(* Logix 5000 project; controller CarbonScout_MK6 vendor 1 type 14 code 154 rev 32.11; software revision 32.00; part 8 of 17 *)
(* tags used below, declared in another part *)
   AI_AIT_01 : P_AIn;   // pH
   AI_AIT_02 : P_AIn;   // DO
   AI_Booster : P_AIn;   // Booster Tank Level
   AI_FIT_01 : P_AIn;   // Purge water flow
   AI_LIT_01 : P_AIn;   // Carbon Scout Laser Level Transmitter
   AI_LIT_02 : P_AIn;   // Carbon Scout Cone Level Transmitter
   AI_PIT_01 : P_AIn;   // Water supply pressure
   AI_TIT_01 : P_AIn;   // Temperature
   AI_WIT_01 : P_AIn;   // Weight measure
   Client_to_Gekko : DINT[10];
   CS_Alarms : P_Alarm[80];
   CS_DINTParams : DINT[100];
   CS_REALParams : REAL[80];   // CS REAL Parameters
   CS_Result : CS_Results;   // Sample Result Live Async
   CS_SampleSeq : DINT[129];
   CS_Seq : GEK_Sequence;
   CS_Seq_ControlStop : BOOL;
   CS_Seq_CrashStop : BOOL;
   CS_STRINGParams : STRING_20[10];
   CS_Tank : CS_TankParams[20];

        As_Model[1].A := 1.0, Se_ErrRaw := 1.0, Se_Model[0].A := 1.0, Se_Model[1].A := 1.0, Rb_ErrRaw := 2.0, Rb_Model[0].A := 1.0, Rb_Model[1].A := 1.0, Sr_Raw := 7.0, Sr_ErrRaw := 1.0, Sr_Model[0].A := 1.0, Sr_Model[1].A := 1.0, Y_ErrRaw := 3.0, Y_Model[0].A := 1.0, Y_Model[1].A := 1.0, Zr_Raw := 7.0, Zr_ErrRaw := 1.0, Zr_Model[0].A := 1.0, Zr_Model[1].A := 1.0, Nb_ErrRaw := 3.0, Nb_Model[0].A := 1.0, Nb_Model[1].A := 1.0, Mo_Raw := 80.0, Mo_ErrRaw := 2.0, Mo_Model[0].A := 1.0, Mo_Model[1].A := 1.0, Ag_ErrRaw := 137.0, Ag_Model[0].A := 1.0, Ag_Model[1].A := 1.0, Cd_ErrRaw := 12.0, Cd_Model[0].A := 1.0, Cd_Model[1].A := 1.0, Sn_ErrRaw := 15.0, Sn_Model[0].A := 1.0, Sn_Model[1].A := 1.0, Sb_ErrRaw := 20.0, Sb_Model[0].A := 1.0, Sb_Model[1].A := 1.0, Ba_Model[0].A := 1.0, Ba_Model[1].A := 1.0, La_Model[0].A := 1.0, La_Model[1].A := 1.0, Ce_Model[0].A := 1.0, Ce_Model[1].A := 1.0, Pr_Model[0].A := 1.0, Pr_Model[1].A := 1.0, Nd_Model[0].A := 1.0, Nd_Model[1].A := 1.0, W_ErrRaw := 13.0, W_Model[0].A := 1.0, W_Model[1].A := 1.0, Hg_ErrRaw := 7.0, Hg_Model[0].A := 1.0, Hg_Model[1].A := 1.0, Pb_ErrRaw := 3.0, Pb_Model[0].A := 1.0, Pb_Model[1].A := 1.0, Bi_ErrRaw := 22.0, Bi_Model[0].A := 1.0, Bi_Model[1].A := 1.0, Th_Raw := 30.0,
        Th_ErrRaw := 4.0, Th_Model[0].A := 1.0, Th_Model[1].A := 1.0, U_Raw := 18.0, U_ErrRaw := 2.0, U_Model[0].A := 1.0, U_Model[1].A := 1.0, LE_Model[0].A := 1.0, LE_Model[1].A := 1.0); {access Read Only}
   CS_XRF_ProbeTemp : REAL := 35.0;
   CS_XRF_RawModel : REAL[4] := ([0] := -92.85, [1] := 5.88, [2] := -0.00666);
        [3]   // Thrid Coefficent
        [1]   // First cooefficent
        [2]   // Second Coefficent
        [0]   // Intercept
   Data_Alarm1 : DINT;
        .3   // Purge Water Flow Low CNT reached
        .25   // Check Tank diagnostics
        .24   // Hopper Levels Not OK at the Start Alarm
        .0   // Low Air Pressure Alarm
        .1   // Purge Water Flow Alarm
        .30   // XRF HW Error
        .10   // Tank 7 Offline Alarm
        .15   // Solution fill time exceeded Tank 2
        .14   // Solution fill time exceeded Tank 1
        .11   // Tank 8 Offline Alarm
        .16   // Solution fill time exceeded Tank 3
        .17   // Solution fill time exceeded Tank 4
        .4   // Tank 1 Offline Alarm
        .5   // Tank 2 Offline Alarm
        .6   // Tank 3 Offline Alarm
        .7   // Tank 4 Offline Alarm
        .8   // Tank 5 Offline Alarm
        .18   // Solution fill time exceeded Tank 5
        .13   // Tank 10 Offline Alarm
        .12   // Tank 9 Offline Alarm
        .28   // XRF User Abord Alarm
        .2   // No Available Tank Alarm
        .29   // XRF heartbeat fault
        .9   // Tank 6 Offline Alarm
        .19   // Solution fill time exceeded Tank 6
        .20   // Solution fill time exceeded Tank 7
        .21   // Solution fill time exceeded Tank 8
        .22   // Solution fill time exceeded Tank 9
        .23   // Solution fill time exceeded Tank 10
        .31   // Reserved Do Not Use
        .26   // Spare
        .27   // Spare
   Data_Alarm2 : DINT := 3072;
        .25   // Solution fill time exceeded Tank 11
        .2   // XRF Interlock Lid or E-stop
        .9   // XRF Instrument Not fully in workstation
        .4   // XRF External Interlock Abort
        .7   // XRF Exposure Lasted Longer THan Expected
        .6   // XRF No Counts In Spectrum
        .26   // Solution fill time exceeded Tank 12
        .27   // Solution fill time exceeded Tank 13
        .28   // Solution fill time exceeded Tank 14
        .29   // Solution fill time exceeded Tank 15
        .30   // Solution fill time exceeded Tank 16
        .12   // Laser Compartment Dirty Alarm
        .0   // XRF Trigger Released
        .3   // XRF Proximity Failure (Air Shoot)
        .5   // XRF No longer Needed
        .1   // XRF HW Watchdog Timeout
        .19   // Tank 11 Offline Alarm
        .20   // Tank 12 Offline Alarm
        .21   // Tank 13 Offline Alarm
        .22   // Tank 14 Offline Alarm
        .23   // Tank 15 Offline Alarm
        .24   // Tank 16 Offline Alarm
        .31   // Reserved Do Not Use
        .10   // Spare
        .11   // Spare
        .13   // Spare
        .14   // Spare
        .15   // Spare
        .16   // Spare
        .17   // Spare
        .18   // Spare
        .8   // XRF Proximity Abort
   Data_Alarm3 : DINT;
        .6   // Laser High Fluctuation Alarm
        .4   // Water Supply Line Leak
        .7   // Line Leak
        .3   // Valve Maintenance Request Alarm
        .31   // Reserved Do Not Use
        .9   // Radar cal Not Done
        .10   // Spare
        .1   // Sample Line Break
        .0   // Sample Line Blocked
        .8   // XRF door opened
        .11   // Spare
        .12   // Spare
        .13   // Spare
        .5   // Pegged Screen Alarm
        .14   // Spare
        .15   // Spare
        .16   // Spare
        .17   // Spare
        .18   // Spare
        .19   // Spare
        .20   // Spare
        .21   // Spare
        .22   // Spare
        .23   // Spare
        .24   // Spare
        .25   // Spare
        .26   // Spare
        .27   // Spare
        .28   // Spare
        .29   // Spare
        .30   // Spare
        .2   // Sample Cone Dirty Alarm (Density is not 1)
   Data_constant1 : BOOL := 1;
   Data_Saved : BOOL;
   Data_Saver : BOOL := 1;
   Data_Trigger : BOOL;
   Data_Triggered : BOOL;
   Delete2_Trigger : BOOL;
   Delete_Trigger : BOOL;
   DOL_Booster_Fault : BOOL;
   DOL_Discharge_Fault : BOOL;
   Email_Trigger : BOOL;
   Email_Trigger2 : BOOL;
   FOQ01 : TOTALIZER := (Gain := 1.0, Target := 1000.0, ProgProgReq := 1, ProgStopReq := 1, ProgResetReq := 1, RTSTime := 1, ProgOper := 1, ProgResetDone := 1, LowInCutoffFlag := 1, DeltaT := 0.1);   // PurgeTotaliser
   FOQ02 : TOTALIZER := (Gain := 1.0, Target := 5.0, ProgProgReq := 1, ProgStopReq := 1, ProgResetReq := 1, RTSTime := 1, ProgOper := 1, ProgResetDone := 1, LowInCutoffFlag := 1, DeltaT := 0.1);   // Radar Calibration Totaliser
   Gekko_to_Client : DINT[10] := ([0] := 2081, [1] := 240);
   LeakCheck : BOOL;
   N50 : DINT[20] := ([0] := 196608, [2] := 6, [3] := 12, [4] := 9, [5] := 39, [6] := 1447, [8] := -11, [13] := 1, [14] := 986); {access Read Only}   // Out To Client (Ready only)
        [14]   // HeartBeat Increment 4sec
        [0].10   // XV11
        [0].0   // XV01
        [0].1   // XV02
        [0].2   // XV03
        [0].3   // XV04
        [0].11   // XV12
        [0].4   // XV05
        [0].5   // XV06
        [0].12   // Xv13
        [3]   // Seq intlk/Perm
        [0].6   // XV07
        [0].7   // XV08
        [0].13   // xV14
        [0].14   // xv15
        [0].15   // xv16
        [0].19   // xv21_30
        [12]   // Active Step
        [11]   // DIST
        [0].16   // xv17
        [0].27   // SPR01
        [0].17   // xv18
        [0].18   // xv19
        [0].20   // xv30
        [0].21   // xv31
        [0].22   // xv32
        [0].23   // xv33
        [0].24   // xv34
        [0].25   // xv35
        [0].26   // xv36
        [9]   // XRF
        [1]   // Time Elapsed
        [2]   // Current Tank
        [0].8   // XV09
        [4]   // AIT01
        [5]   // AIT02
        [6]   // LIT01
        [7]   // LIT02
        [8]   // WIT01
        [0].9   // XV10
        [0]   // Valve Out
        [10]   // CN
        [13].1   // External Interlock enabled
        [13].0   // Heart bead 1 second
        [13]   // BOOLS Digital Status
   N51 : DINT[5] := ([1] := 9);   // From Client
        [0].2   // Remote Auto/Man Request 1 = Auto, 0 = Man
        [0]   // Command
        [1]   // remote Tank Number Request
        [0].5   // Remote /Local 0 = Local 1= Remote
        [0].3   // Tank Hold
        [0].4   // Reset All
        [0].1   // Control Stop
        [0].0   // Start
   NetworkHealthy : DINT := -2147483645;
        .0   // Valve Module Healthy 1= failed 0= healthy
        .31   // Proceed Network Checking Flag
        .1   // DO PH Module Healthy 1= failed 0= healthy
   Oneshot : DINT := 17308672;
   Oneshot2 : DINT := 155189248;
   Oneshot3 : DINT := 10;
   PLC_Powered : BOOL;
   Powered_Up : TIMER := (PRE := 1000);
   Reg_Cal : REAL[10] := ([0] := 1810.0, [1] := 2500.0, [2] := 4525000.0, [3] := 3276100.0, [4] := 6250000.0, [5] := 1.4964869, [6] := 1.4392458, [7] := 2.1538124, [8] := 833447.3, [9] := 1562500.0);   // working calculation variables
        [0]   // x
        [1]   // y
        [2]   // xy
        [3]   // x*x
        [4]   // y*y
        [5]   // zx
        [6]   // zy
        [7]   // zx*zy
        [8]   // x-xavg*x-xavg
        [9]   // y-yavg*y-yavg
   Reg_Calsum : REAL[10] := ([0] := 26912.0, [1] := 37500.0, [2] := 48968000.0, [3] := 34934564.0, [4] := 68750000.0, [5] := 4.7683716e-07, [6] := -2.3841858e-07, [7] := 28.929726, [8] := 10792706.0, [9] := 21875000.0);   // running sum of calc variables
        [0]   // x
        [1]   // y
        [2]   // xy
        [3]   // x*x
        [4]   // y*y
        [5]   // zx
        [6]   // zy
        [7]   // zx*zy
        [8]   // x-xavg*x-xavg
        [9]   // y-yavg*y-yavg
   Reg_DINTparams : DINT[8] := ([1] := 3, [2] := 30, [3] := 29, [4] := 28, [6] := 3, [7] := 7247);   // Dint and bools for calcs
        [1]   // cal cycle
        [2]   // sample number
        [3]   // sample number -1
        [4]   // sample number -2
        [6]   // bools and oneshots
        [6].0   // enable Low to high will start calc
        [6].1   // oneshot
        [6].2   // oneshot
        [7]   // calflags
        [7].0   // 1st sum done
        [7].1   // 2nd sum done
        [7].10   // Standard error acceptable
        [7].2   // 3rd sum done
        [7].3   // 4th sum done
        [7].4   // Status Calculating
        [7].5   // Skip index
        [7].6   // R squared acceptable
        [7].7   // HMI calculate Bool
        [7].8   // HMI accept new model
        [7].11   // Model accepted and waiting for recaculation
        [7].12   // HMI accept button inhibit visability 1= Visable and not clickable
   Reg_InX : REAL[30] := ([1] := 2.0, [2] := 3.0, [3] := 2.0, [4] := 2.0, [5] := 381.0, [6] := 392.0, [7] := 382.0, [8] := 352.0, [9] := 393.0, [10] := 741.0, [11] := 745.0, [12] := 760.0, [13] := 763.0, [14] := 803.0, [15] := 1070.0, [16] := 1053.0, [17] := 1062.0, [18] := 986.0, [19] := 1052.0, [20] := 1477.0, [21] := 1421.0, [22] := 1377.0, [23] := 1422.0, [24] := 1400.0, [25] := 1682.0, [26] := 1698.0, [27] := 1843.0, [28] := 1838.0, [29] := 1810.0);   // X input for calcs
   Reg_InY : REAL[30] := ([5] := 500.0, [6] := 500.0, [7] := 500.0, [8] := 500.0, [9] := 500.0, [10] := 1000.0, [11] := 1000.0, [12] := 1000.0, [13] := 1000.0, [14] := 1000.0, [15] := 1500.0, [16] := 1500.0, [17] := 1500.0, [18] := 1500.0, [19] := 1500.0, [20] := 2000.0, [21] := 2000.0, [22] := 2000.0, [23] := 2000.0, [24] := 2000.0, [25] := 2500.0, [26] := 2500.0, [27] := 2500.0, [28] := 2500.0, [29] := 2500.0);   // Y input for pairs
   Reg_Model : REAL[4] := ([0] := -48.061447, [1] := 2.2187226, [3] := 1.0);   // Calculated model output and site model
        [0]   // Holding site int
        [1]   // Holding site 1st
        [2]   // Site int
        [3]   // Site 1st
   Reg_Out : REAL[14] := ([0] := -24.030724, [1] := 1.4202185, [2] := 897.06665, [3] := 1250.0, [4] := 610.051, [5] := 868.51044, [6] := 0.9975768, [7] := 0.99515945, [8] := 372162.28, [9] := 754310.4, [10] := 0.9949866, [11] := 61.495235);   // Output of calculation
        [0]   // a
        [10]   // r*r adjusted
        [11]   // Standard Error
        [1]   // b
        [2]   // xavg
        [3]   // yavg
        [4]   // sdx s
        [5]   // sdy s
        [6]   // r
        [7]   // r*r
        [8]   // SUM(x-xavg*x-xavg)/N-1
        [9]   // SUM(y-yavg*y-yavg)/N-1
   Simulation : DINT;
        .0   // SP skipping simulation
        .6   // Email trigger sim
        .5   // Data save Sim
        .8   // Discharge Sim
        .2   // XRF simulation
        .3   // CN SIM
        .1   // Instrument Simulation
        .7   // Booster Sim
   TankNum : DINT := 6;
   TankPointer : DINT := 5;
   test : DINT;
   TimeAndDate : DINT[7] := ([0] := 1998, [1] := 6, [2] := 27, [3] := 19, [4] := 1, [5] := 9, [6] := 869613);
        [2]   // Day
        [0]   // Year
        [6]   // Millisecond
        [4]   // Minute
        [3]   // Hour
        [5]   // Second
        [1]   // Month
   TimeAndDateW : DINT[7] := ([0] := 2021, [1] := 6, [2] := 7, [3] := 13, [4] := 23);
   Uptime : DINT := 8453;   // sec
   Valve_Booster1 : P_ValveSO := (Inp_PermOK := 1, Inp_NBPermOK := 1, Inp_IntlkOK := 1, Inp_NBIntlkOK := 1, Cfg_LSFail := 1, Cfg_ProgDefault := 1, Cfg_ShedOnFullStall := 1, Cfg_ShedOnTransitStall := 1, Cfg_ShedOnIOFault := 1, Cfg_FullStallAckReqd := 1, Cfg_TransitStallAckReqd := 1, Cfg_IntlkTripAckReqd := 1, Cfg_IOFaultAckReqd := 1, Cfg_FullStallSeverity := 1000, Cfg_TransitStallSeverity := 1000, Cfg_IntlkTripSeverity := 500, Cfg_IOFaultSeverity := 1000, Cfg_SimFdbkT := 2, Cfg_FullStallT := 5, Cfg_TransitStallT := 10, PCmd_Acq := 1, SrcQ_IO := 2, SrcQ := 2, Val_Fdbk := 1, Val_Sts := 1, Val_Mode := 8, Sts_Closed := 1, Sts_Available := 1, Sts_Prog := 1, Ack_FullStall := 1, Ack_TransitStall := 1, Ack_IntlkTrip := 1, Ack_IOFault := 1, Rdy_Bypass := 1);   // Booster Top Up Valve
   Valve_Discharge1 : P_ValveSO := (Inp_PermOK := 1, Inp_NBPermOK := 1, Inp_IntlkOK := 1, Inp_NBIntlkOK := 1, Cfg_LSFail := 1, Cfg_ProgDefault := 1, Cfg_ShedOnFullStall := 1, Cfg_ShedOnTransitStall := 1, Cfg_ShedOnIOFault := 1, Cfg_FullStallAckReqd := 1, Cfg_TransitStallAckReqd := 1, Cfg_IntlkTripAckReqd := 1, Cfg_IOFaultAckReqd := 1, Cfg_FullStallSeverity := 1000, Cfg_TransitStallSeverity := 1000, Cfg_IntlkTripSeverity := 500, Cfg_IOFaultSeverity := 1000, Cfg_SimFdbkT := 2, Cfg_FullStallT := 5, Cfg_TransitStallT := 10, PCmd_Close := 1, PCmd_Acq := 1, SrcQ_IO := 2, SrcQ := 2, Val_Fdbk := 1, Val_Sts := 1, Val_Mode := 8, Sts_Closed := 1, Sts_Available := 1, Sts_Prog := 1, Ack_FullStall := 1, Ack_TransitStall := 1, Ack_IntlkTrip := 1, Ack_IOFault := 1, Rdy_Bypass := 1);   // Top Up Valve
   Valve_Discharge2 : P_ValveSO := (Inp_PermOK := 1, Inp_NBPermOK := 1, Inp_IntlkOK := 1, Inp_NBIntlkOK := 1, Cfg_LSFail := 1, Cfg_ProgDefault := 1, Cfg_ShedOnFullStall := 1, Cfg_ShedOnTransitStall := 1, Cfg_ShedOnIOFault := 1, Cfg_FullStallAckReqd := 1, Cfg_TransitStallAckReqd := 1, Cfg_IntlkTripAckReqd := 1, Cfg_IOFaultAckReqd := 1, Cfg_FullStallSeverity := 1000, Cfg_TransitStallSeverity := 1000, Cfg_IntlkTripSeverity := 500, Cfg_IOFaultSeverity := 1000, Cfg_SimFdbkT := 2, Cfg_FullStallT := 5, Cfg_TransitStallT := 10, PCmd_Close := 1, PCmd_Acq := 1, SrcQ_IO := 2, SrcQ := 2, Val_Fdbk := 1, Val_Sts := 1, Val_Mode := 8, Sts_Closed := 1, Sts_Available := 1, Sts_Prog := 1, Ack_FullStall := 1, Ack_TransitStall := 1, Ack_IntlkTrip := 1, Ack_IOFault := 1, Rdy_Bypass := 1);   // Discharge Valve
   Valve_SPR_01 : P_ValveSO := (Inp_PermOK := 1, Inp_NBPermOK := 1, Inp_IntlkOK := 1, Inp_NBIntlkOK := 1, Cfg_LSFail := 1, Cfg_ProgDefault := 1, Cfg_ShedOnFullStall := 1, Cfg_ShedOnTransitStall := 1, Cfg_ShedOnIOFault := 1, Cfg_FullStallAckReqd := 1, Cfg_TransitStallAckReqd := 1, Cfg_IntlkTripAckReqd := 1, Cfg_IOFaultAckReqd := 1, Cfg_FullStallSeverity := 1000, Cfg_TransitStallSeverity := 1000, Cfg_IntlkTripSeverity := 500, Cfg_IOFaultSeverity := 1000, Cfg_FullStallT := 5, Cfg_TransitStallT := 10, PCmd_Close := 1, PCmd_Acq := 1, SrcQ_IO := 2, SrcQ := 2, Val_Fdbk := 1, Val_Sts := 1, Val_Mode := 8, Sts_Closed := 1, Sts_Available := 1, Sts_Prog := 1, Ack_FullStall := 1, Ack_TransitStall := 1, Ack_IntlkTrip := 1, Ack_IOFault := 1, Rdy_Bypass := 1);   // Air injection valve
   Valve_SPR_01_Stats : GekkoValveStat := (Inp_Closed := 1, Out_CloseCNT := 21352.0, Inp_OpenCNTSP := 9999999.0, Out_CloseReached := 1);
   Valve_XV_01 : P_ValveSO := (Inp_PermOK := 1, Inp_NBPermOK := 1, Inp_IntlkOK := 1, Inp_NBIntlkOK := 1, Cfg_LSFail := 1, Cfg_ProgDefault := 1, Cfg_ShedOnFullStall := 1, Cfg_ShedOnTransitStall := 1, Cfg_ShedOnIOFault := 1, Cfg_FullStallAckReqd := 1, Cfg_TransitStallAckReqd := 1, Cfg_IntlkTripAckReqd := 1, Cfg_IOFaultAckReqd := 1, Cfg_FullStallSeverity := 1000, Cfg_TransitStallSeverity := 1000, Cfg_IntlkTripSeverity := 500, Cfg_IOFaultSeverity := 1000, Cfg_FullStallT := 5, Cfg_TransitStallT := 10, PCmd_Close := 1, PCmd_Acq := 1, SrcQ_IO := 2, SrcQ := 2, Val_Fdbk := 1, Val_Sts := 1, Val_Mode := 8, Sts_Closed := 1, Sts_Available := 1, Sts_Prog := 1, Ack_FullStall := 1, Ack_TransitStall := 1, Ack_IntlkTrip := 1, Ack_IOFault := 1, Rdy_Bypass := 1);   // Sample Valve Tank 1
   Valve_XV_01_Stats : GekkoValveStat := (Inp_Closed := 1, Out_OpenCNT := 1549.0, Out_CloseCNT := 5694.0, Inp_OpenCNTSP := 5000.0, Out_CloseReached := 1);
   Valve_XV_02 : P_ValveSO := (Inp_PermOK := 1, Inp_NBPermOK := 1, Inp_IntlkOK := 1, Inp_NBIntlkOK := 1, Cfg_LSFail := 1, Cfg_ProgDefault := 1, Cfg_ShedOnFullStall := 1, Cfg_ShedOnTransitStall := 1, Cfg_ShedOnIOFault := 1, Cfg_FullStallAckReqd := 1, Cfg_TransitStallAckReqd := 1, Cfg_IntlkTripAckReqd := 1, Cfg_IOFaultAckReqd := 1, Cfg_FullStallSeverity := 1000, Cfg_TransitStallSeverity := 1000, Cfg_IntlkTripSeverity := 500, Cfg_IOFaultSeverity := 1000, Cfg_FullStallT := 5, Cfg_TransitStallT := 10, PCmd_Close := 1, PCmd_Acq := 1, SrcQ_IO := 2, SrcQ := 2, Val_Fdbk := 1, Val_Sts := 1, Val_Mode := 8, Sts_Closed := 1, Sts_Available := 1, Sts_Prog := 1, Ack_FullStall := 1, Ack_TransitStall := 1, Ack_IntlkTrip := 1, Ack_IOFault := 1, Rdy_Bypass := 1);   // Sample Valve Tank 2
   Valve_XV_02_Stats : GekkoValveStat := (Inp_Closed := 1, Out_OpenCNT := 1166.0, Out_CloseCNT := 5225.0, Inp_OpenCNTSP := 5000.0, Out_CloseReached := 1);
   Valve_XV_03 : P_ValveSO := (Inp_PermOK := 1, Inp_NBPermOK := 1, Inp_IntlkOK := 1, Inp_NBIntlkOK := 1, Cfg_LSFail := 1, Cfg_ProgDefault := 1, Cfg_ShedOnFullStall := 1, Cfg_ShedOnTransitStall := 1, Cfg_ShedOnIOFault := 1, Cfg_HasIntlkTripAlm := 1, Cfg_HasIOFaultAlm := 1, Cfg_IntlkTripAckReqd := 1, Cfg_FullStallSeverity := 1000, Cfg_TransitStallSeverity := 1000, Cfg_IntlkTripSeverity := 500, Cfg_IOFaultSeverity := 1000, Cfg_FullStallT := 5, Cfg_TransitStallT := 10, PCmd_Close := 1, PCmd_Acq := 1, SrcQ_IO := 2, SrcQ := 2, Val_Fdbk := 1, Val_Sts := 1, Val_Mode := 8, Sts_Closed := 1, Sts_Available := 1, Sts_Prog := 1, Ack_FullStall := 1, Ack_TransitStall := 1, Ack_IntlkTrip := 1, Ack_IOFault := 1, Rdy_Bypass := 1);   // Sample Valve Tank 3
   Valve_XV_03_Stats : GekkoValveStat := (Inp_Closed := 1, Out_OpenCNT := 1129.0, Out_CloseCNT := 4654.0, Inp_OpenCNTSP := 5000.0, Out_CloseReached := 1);
   Valve_XV_04 : P_ValveSO := (Inp_PermOK := 1, Inp_NBPermOK := 1, Inp_IntlkOK := 1, Inp_NBIntlkOK := 1, Cfg_LSFail := 1, Cfg_ProgDefault := 1, Cfg_ShedOnFullStall := 1, Cfg_ShedOnTransitStall := 1, Cfg_ShedOnIOFault := 1, Cfg_FullStallAckReqd := 1, Cfg_TransitStallAckReqd := 1, Cfg_IntlkTripAckReqd := 1, Cfg_IOFaultAckReqd := 1, Cfg_FullStallSeverity := 1000, Cfg_TransitStallSeverity := 1000, Cfg_IntlkTripSeverity := 500, Cfg_IOFaultSeverity := 1000, Cfg_FullStallT := 5, Cfg_TransitStallT := 10, PCmd_Close := 1, PCmd_Acq := 1, SrcQ_IO := 2, SrcQ := 2, Val_Fdbk := 1, Val_Sts := 1, Val_Mode := 8, Sts_Closed := 1, Sts_Available := 1, Sts_Prog := 1, Ack_FullStall := 1, Ack_TransitStall := 1, Ack_IntlkTrip := 1, Ack_IOFault := 1, Rdy_Bypass := 1);   // Sample Valve Tank 4
   Valve_XV_04_Stats : GekkoValveStat := (Inp_Closed := 1, Out_OpenCNT := 1127.0, Out_CloseCNT := 4762.0, Inp_OpenCNTSP := 5000.0, Out_CloseReached := 1);
   Valve_XV_05 : P_ValveSO := (Inp_PermOK := 1, Inp_NBPermOK := 1, Inp_IntlkOK := 1, Inp_NBIntlkOK := 1, Cfg_LSFail := 1, Cfg_ProgDefault := 1, Cfg_ShedOnFullStall := 1, Cfg_ShedOnTransitStall := 1, Cfg_ShedOnIOFault := 1, Cfg_FullStallAckReqd := 1, Cfg_TransitStallAckReqd := 1, Cfg_IntlkTripAckReqd := 1, Cfg_IOFaultAckReqd := 1, Cfg_FullStallSeverity := 1000, Cfg_TransitStallSeverity := 1000, Cfg_IntlkTripSeverity := 500, Cfg_IOFaultSeverity := 1000, Cfg_FullStallT := 5, Cfg_TransitStallT := 10, PCmd_Close := 1, PCmd_Acq := 1, SrcQ_IO := 2, SrcQ := 2, Val_Fdbk := 1, Val_Sts := 1, Val_Mode := 8, Sts_Closed := 1, Sts_Available := 1, Sts_Prog := 1, Ack_FullStall := 1, Ack_TransitStall := 1, Ack_IntlkTrip := 1, Ack_IOFault := 1, Rdy_Bypass := 1);   // Sample Valve Tank 5
   Valve_XV_05_Stats : GekkoValveStat := (Inp_Closed := 1, Out_OpenCNT := 1115.0, Out_CloseCNT := 4670.0, Inp_OpenCNTSP := 5000.0, Out_CloseReached := 1);
   Valve_XV_06 : P_ValveSO := (Inp_PermOK := 1, Inp_NBPermOK := 1, Inp_IntlkOK := 1, Inp_NBIntlkOK := 1, Cfg_LSFail := 1, Cfg_ProgDefault := 1, Cfg_ShedOnFullStall := 1, Cfg_ShedOnTransitStall := 1, Cfg_ShedOnIOFault := 1, Cfg_FullStallAckReqd := 1, Cfg_TransitStallAckReqd := 1, Cfg_IntlkTripAckReqd := 1, Cfg_IOFaultAckReqd := 1, Cfg_FullStallSeverity := 1000, Cfg_TransitStallSeverity := 1000, Cfg_IntlkTripSeverity := 500, Cfg_IOFaultSeverity := 1000, Cfg_FullStallT := 5, Cfg_TransitStallT := 10, PCmd_Close := 1, PCmd_Acq := 1, SrcQ_IO := 2, SrcQ := 2, Val_Fdbk := 1, Val_Sts := 1, Val_Mode := 8, Sts_Closed := 1, Sts_Available := 1, Sts_Prog := 1, Ack_FullStall := 1, Ack_TransitStall := 1, Ack_IntlkTrip := 1, Ack_IOFault := 1, Rdy_Bypass := 1);   // Sample Valve Tank 6
   Valve_XV_06_Stats : GekkoValveStat := (Inp_Closed := 1, Out_OpenCNT := 1086.0, Out_CloseCNT := 4737.0, Inp_OpenCNTSP := 5000.0, Out_CloseReached := 1);
   Valve_XV_07 : P_ValveSO := (Inp_PermOK := 1, Inp_NBPermOK := 1, Inp_IntlkOK := 1, Inp_NBIntlkOK := 1, Cfg_LSFail := 1, Cfg_ProgDefault := 1, Cfg_ShedOnFullStall := 1, Cfg_ShedOnTransitStall := 1, Cfg_ShedOnIOFault := 1, Cfg_FullStallAckReqd := 1, Cfg_TransitStallAckReqd := 1, Cfg_IntlkTripAckReqd := 1, Cfg_IOFaultAckReqd := 1, Cfg_FullStallSeverity := 1000, Cfg_TransitStallSeverity := 1000, Cfg_IntlkTripSeverity := 500, Cfg_IOFaultSeverity := 1000, Cfg_FullStallT := 5, Cfg_TransitStallT := 10, PCmd_Close := 1, PCmd_Acq := 1, SrcQ_IO := 2, SrcQ := 2, Val_Fdbk := 1, Val_Sts := 1, Val_Mode := 8, Sts_Closed := 1, Sts_Available := 1, Sts_Prog := 1, Ack_FullStall := 1, Ack_TransitStall := 1, Ack_IntlkTrip := 1, Ack_IOFault := 1, Rdy_Bypass := 1);   // Sample Valve Tank 7
   Valve_XV_07_Stats : GekkoValveStat := (Inp_Closed := 1, Out_OpenCNT := 1068.0, Out_CloseCNT := 4641.0, Inp_OpenCNTSP := 5000.0, Out_CloseReached := 1);
   Valve_XV_08 : P_ValveSO := (Inp_PermOK := 1, Inp_NBPermOK := 1, Inp_IntlkOK := 1, Inp_NBIntlkOK := 1, Cfg_LSFail := 1, Cfg_ProgDefault := 1, Cfg_ShedOnFullStall := 1, Cfg_ShedOnTransitStall := 1, Cfg_ShedOnIOFault := 1, Cfg_FullStallAckReqd := 1, Cfg_TransitStallAckReqd := 1, Cfg_IntlkTripAckReqd := 1, Cfg_IOFaultAckReqd := 1, Cfg_FullStallSeverity := 1000, Cfg_TransitStallSeverity := 1000, Cfg_IntlkTripSeverity := 500, Cfg_IOFaultSeverity := 1000, Cfg_FullStallT := 5, Cfg_TransitStallT := 10, PCmd_Close := 1, PCmd_Acq := 1, SrcQ_IO := 2, SrcQ := 2, Val_Fdbk := 1, Val_Sts := 1, Val_Mode := 8, Sts_Closed := 1, Sts_Available := 1, Sts_Prog := 1, Ack_FullStall := 1, Ack_TransitStall := 1, Ack_IntlkTrip := 1, Ack_IOFault := 1, Rdy_Bypass := 1);   // Sample Valve Tank 8
   Valve_XV_08_Stats : GekkoValveStat := (Inp_Closed := 1, Out_OpenCNT := 1057.0, Out_CloseCNT := 4478.0, Inp_OpenCNTSP := 5000.0, Out_CloseReached := 1);
   Valve_XV_09 : P_ValveSO := (Inp_PermOK := 1, Inp_NBPermOK := 1, Inp_IntlkOK := 1, Inp_NBIntlkOK := 1, Cfg_LSFail := 1, Cfg_ProgDefault := 1, Cfg_ShedOnFullStall := 1, Cfg_ShedOnTransitStall := 1, Cfg_ShedOnIOFault := 1, Cfg_FullStallAckReqd := 1, Cfg_TransitStallAckReqd := 1, Cfg_IntlkTripAckReqd := 1, Cfg_IOFaultAckReqd := 1, Cfg_FullStallSeverity := 1000, Cfg_TransitStallSeverity := 1000, Cfg_IntlkTripSeverity := 500, Cfg_IOFaultSeverity := 1000, Cfg_FullStallT := 5, Cfg_TransitStallT := 10, PCmd_Close := 1, PCmd_Acq := 1, SrcQ_IO := 2, SrcQ := 2, Val_Fdbk := 1, Val_Sts := 1, Val_Mode := 8, Sts_Closed := 1, Sts_Available := 1, Sts_Prog := 1, Ack_FullStall := 1, Ack_TransitStall := 1, Ack_IntlkTrip := 1, Ack_IOFault := 1, Rdy_Bypass := 1);   // Sample Valve Tank 9
   Valve_XV_09_Stats : GekkoValveStat := (Inp_Closed := 1, Out_CloseCNT := 3056.0, Inp_OpenCNTSP := 5000.0, Out_CloseReached := 1);
   Valve_XV_10 : P_ValveSO := (Inp_PermOK := 1, Inp_NBPermOK := 1, Inp_IntlkOK := 1, Inp_NBIntlkOK := 1, Cfg_LSFail := 1, Cfg_ProgDefault := 1, Cfg_ShedOnFullStall := 1, Cfg_ShedOnTransitStall := 1, Cfg_ShedOnIOFault := 1, Cfg_FullStallAckReqd := 1, Cfg_TransitStallAckReqd := 1, Cfg_IntlkTripAckReqd := 1, Cfg_IOFaultAckReqd := 1, Cfg_FullStallSeverity := 1000, Cfg_TransitStallSeverity := 1000, Cfg_IntlkTripSeverity := 500, Cfg_IOFaultSeverity := 1000, Cfg_FullStallT := 5, Cfg_TransitStallT := 10, PCmd_Close := 1, PCmd_Acq := 1, SrcQ_IO := 2, SrcQ := 2, Val_Fdbk := 1, Val_Sts := 1, Val_Mode := 8, Sts_Closed := 1, Sts_Available := 1, Sts_Prog := 1, Ack_FullStall := 1, Ack_TransitStall := 1, Ack_IntlkTrip := 1, Ack_IOFault := 1, Rdy_Bypass := 1);   // Sample Valve Tank 10
   Valve_XV_10_Stats : GekkoValveStat := (Inp_Closed := 1, Out_OpenCNT := 6.0, Out_CloseCNT := 3372.0, Inp_OpenCNTSP := 5000.0, Out_CloseReached := 1);
   Valve_XV_11 : P_ValveSO := (Inp_PermOK := 1, Inp_NBPermOK := 1, Inp_IntlkOK := 1, Inp_NBIntlkOK := 1, Cfg_LSFail := 1, Cfg_ProgDefault := 1, Cfg_ShedOnFullStall := 1, Cfg_ShedOnTransitStall := 1, Cfg_ShedOnIOFault := 1, Cfg_FullStallAckReqd := 1, Cfg_TransitStallAckReqd := 1, Cfg_IntlkTripAckReqd := 1, Cfg_IOFaultAckReqd := 1, Cfg_FullStallSeverity := 1000, Cfg_TransitStallSeverity := 1000, Cfg_IntlkTripSeverity := 500, Cfg_IOFaultSeverity := 1000, Cfg_FullStallT := 5, Cfg_TransitStallT := 10, PCmd_Close := 1, PCmd_Acq := 1, SrcQ_IO := 2, SrcQ := 2, Val_Fdbk := 1, Val_Sts := 1, Val_Mode := 8, Sts_Closed := 1, Sts_Available := 1, Sts_Prog := 1, Ack_FullStall := 1, Ack_TransitStall := 1, Ack_IntlkTrip := 1, Ack_IOFault := 1, Rdy_Bypass := 1);   // Purge Valve
   Valve_XV_11_Stats : GekkoValveStat := (Inp_Closed := 1, Out_OpenCNT := 8599.0, Out_CloseCNT := 41386.0, Inp_OpenCNTSP := 50000.0, Out_CloseReached := 1);
   Valve_XV_12 : P_ValveSO := (Inp_PermOK := 1, Inp_NBPermOK := 1, Inp_IntlkOK := 1, Inp_NBIntlkOK := 1, Cfg_LSFail := 1, Cfg_ProgDefault := 1, Cfg_ShedOnFullStall := 1, Cfg_ShedOnTransitStall := 1, Cfg_ShedOnIOFault := 1, Cfg_FullStallAckReqd := 1, Cfg_TransitStallAckReqd := 1, Cfg_IntlkTripAckReqd := 1, Cfg_IOFaultAckReqd := 1, Cfg_FullStallSeverity := 1000, Cfg_TransitStallSeverity := 1000, Cfg_IntlkTripSeverity := 500, Cfg_IOFaultSeverity := 1000, Cfg_FullStallT := 5, Cfg_TransitStallT := 10, PCmd_Close := 1, PCmd_Acq := 1, SrcQ_IO := 2, SrcQ := 2, Val_Fdbk := 1, Val_Sts := 1, Val_Mode := 8, Sts_Closed := 1, Sts_Available := 1, Sts_Prog := 1, Ack_FullStall := 1, Ack_TransitStall := 1, Ack_IntlkTrip := 1, Ack_IOFault := 1, Rdy_Bypass := 1);   // Slurry inlet vavle
   Valve_XV_12_Stats : GekkoValveStat := (Inp_Closed := 1, Out_OpenCNT := 6181.0, Out_CloseCNT := 30915.0, Inp_OpenCNTSP := 25000.0, Out_CloseReached := 1);
   Valve_XV_13 : P_ValveSO := (Inp_PermOK := 1, Inp_NBPermOK := 1, Inp_IntlkOK := 1, Inp_NBIntlkOK := 1, Cfg_LSFail := 1, Cfg_ProgDefault := 1, Cfg_ShedOnFullStall := 1, Cfg_ShedOnTransitStall := 1, Cfg_ShedOnIOFault := 1, Cfg_FullStallAckReqd := 1, Cfg_TransitStallAckReqd := 1, Cfg_IntlkTripAckReqd := 1, Cfg_IOFaultAckReqd := 1, Cfg_FullStallSeverity := 1000, Cfg_TransitStallSeverity := 1000, Cfg_IntlkTripSeverity := 500, Cfg_IOFaultSeverity := 1000, Cfg_FullStallT := 5, Cfg_TransitStallT := 10, PCmd_Close := 1, PCmd_Acq := 1, SrcQ_IO := 2, SrcQ := 2, Val_Fdbk := 1, Val_Sts := 1, Val_Mode := 8, Sts_Closed := 1, Sts_Available := 1, Sts_Prog := 1, Ack_FullStall := 1, Ack_TransitStall := 1, Ack_IntlkTrip := 1, Ack_IOFault := 1, Rdy_Bypass := 1);   // Sample line vavle
   Valve_XV_13_Stats : GekkoValveStat := (Inp_Closed := 1, Out_OpenCNT := 146.0, Out_CloseCNT := 336.0, Inp_OpenCNTSP := 2600.0, Out_CloseReached := 1);
   Valve_XV_14 : P_ValveSO := (Inp_PermOK := 1, Inp_NBPermOK := 1, Inp_IntlkOK := 1, Inp_NBIntlkOK := 1, Cfg_LSFail := 1, Cfg_ProgDefault := 1, Cfg_ShedOnFullStall := 1, Cfg_ShedOnTransitStall := 1, Cfg_ShedOnIOFault := 1, Cfg_FullStallAckReqd := 1, Cfg_TransitStallAckReqd := 1, Cfg_IntlkTripAckReqd := 1, Cfg_IOFaultAckReqd := 1, Cfg_FullStallSeverity := 1000, Cfg_TransitStallSeverity := 1000, Cfg_IntlkTripSeverity := 500, Cfg_IOFaultSeverity := 1000, Cfg_FullStallT := 5, Cfg_TransitStallT := 10, PCmd_Close := 1, PCmd_Acq := 1, SrcQ_IO := 2, SrcQ := 2, Val_Fdbk := 1, Val_Sts := 1, Val_Mode := 8, Sts_Closed := 1, Sts_Available := 1, Sts_Prog := 1, Ack_FullStall := 1, Ack_TransitStall := 1, Ack_IntlkTrip := 1, Ack_IOFault := 1, Rdy_Bypass := 1);   // Top wash vavle
   Valve_XV_14_Stats : GekkoValveStat := (Inp_Closed := 1, Out_OpenCNT := 5644.0, Out_CloseCNT := 38383.0, Inp_OpenCNTSP := 100000.0, Out_CloseReached := 1);
   Valve_XV_15 : P_ValveSO := (Inp_PermOK := 1, Inp_NBPermOK := 1, Inp_IntlkOK := 1, Inp_NBIntlkOK := 1, Cfg_LSFail := 1, Cfg_ProgDefault := 1, Cfg_ShedOnFullStall := 1, Cfg_ShedOnTransitStall := 1, Cfg_ShedOnIOFault := 1, Cfg_FullStallAckReqd := 1, Cfg_IntlkTripAckReqd := 1, Cfg_IOFaultAckReqd := 1, Cfg_FullStallSeverity := 1000, Cfg_TransitStallSeverity := 1000, Cfg_IntlkTripSeverity := 500, Cfg_IOFaultSeverity := 1000, Cfg_FullStallT := 5, Cfg_TransitStallT := 10, PCmd_Close := 1, PCmd_Acq := 1, SrcQ_IO := 2, SrcQ := 2, Val_Fdbk := 1, Val_Sts := 1, Val_Mode := 8, Sts_Closed := 1, Sts_Available := 1, Sts_Prog := 1, Ack_FullStall := 1, Ack_TransitStall := 1, Ack_IntlkTrip := 1, Ack_IOFault := 1, Rdy_Bypass := 1);   // Bottme wash vavle
   Valve_XV_15_Stats : GekkoValveStat := (Inp_Closed := 1, Out_OpenCNT := 11346.0, Out_CloseCNT := 65531.0, Inp_OpenCNTSP := 100000.0, Out_CloseReached := 1);
   Valve_XV_16 : P_ValveSO := (Inp_PermOK := 1, Inp_NBPermOK := 1, Inp_IntlkOK := 1, Inp_NBIntlkOK := 1, Cfg_LSFail := 1, Cfg_ProgDefault := 1, Cfg_ShedOnFullStall := 1, Cfg_ShedOnTransitStall := 1, Cfg_ShedOnIOFault := 1, Cfg_FullStallAckReqd := 1, Cfg_TransitStallAckReqd := 1, Cfg_IntlkTripAckReqd := 1, Cfg_IOFaultAckReqd := 1, Cfg_FullStallSeverity := 1000, Cfg_TransitStallSeverity := 1000, Cfg_IntlkTripSeverity := 500, Cfg_IOFaultSeverity := 1000, Cfg_FullStallT := 5, Cfg_TransitStallT := 10, PCmd_Close := 1, PCmd_Acq := 1, SrcQ_IO := 2, SrcQ := 2, Val_Fdbk := 1, Val_Sts := 1, Val_Mode := 8, Sts_Closed := 1, Sts_Available := 1, Sts_Prog := 1, Ack_FullStall := 1, Ack_TransitStall := 1, Ack_IntlkTrip := 1, Ack_IOFault := 1, Rdy_Bypass := 1);   // Potable water valve / Supply Water Valve
   Valve_XV_16_Stats : GekkoValveStat := (Inp_Closed := 1, Out_OpenCNT := 5598.0, Out_CloseCNT := 25174.0, Inp_OpenCNTSP := 100000.0, Out_CloseReached := 1);
   Valve_XV_17 : P_ValveSO := (Inp_PermOK := 1, Inp_NBPermOK := 1, Inp_IntlkOK := 1, Inp_NBIntlkOK := 1, Cfg_FailOpen := 1, Cfg_LSFail := 1, Cfg_ProgDefault := 1, Cfg_ShedOnFullStall := 1, Cfg_ShedOnTransitStall := 1, Cfg_ShedOnIOFault := 1, Cfg_FullStallAckReqd := 1, Cfg_TransitStallAckReqd := 1, Cfg_IntlkTripAckReqd := 1, Cfg_IOFaultAckReqd := 1, Cfg_FullStallSeverity := 1000, Cfg_TransitStallSeverity := 1000, Cfg_IntlkTripSeverity := 500, Cfg_IOFaultSeverity := 1000, Cfg_FullStallT := 5, Cfg_TransitStallT := 10, PCmd_Close := 1, PCmd_Acq := 1, Out := 1, SrcQ_IO := 2, SrcQ := 2, Val_Fdbk := 1, Val_Sts := 1, Val_Mode := 8, Sts_Closed := 1, Sts_Available := 1, Sts_Prog := 1, Ack_FullStall := 1, Ack_TransitStall := 1, Ack_IntlkTrip := 1, Ack_IOFault := 1, Rdy_Bypass := 1);   // Sample cone outlet vavle
   Valve_XV_17_Stats : GekkoValveStat := (Inp_Closed := 1, Out_OpenCNT := 8748.0, Out_CloseCNT := 48939.0, Inp_OpenCNTSP := 50000.0, Out_CloseReached := 1);
   Valve_XV_18 : P_ValveSO := (Inp_PermOK := 1, Inp_NBPermOK := 1, Inp_IntlkOK := 1, Inp_NBIntlkOK := 1, Cfg_FailOpen := 1, Cfg_LSFail := 1, Cfg_ProgDefault := 1, Cfg_ShedOnFullStall := 1, Cfg_ShedOnTransitStall := 1, Cfg_ShedOnIOFault := 1, Cfg_FullStallAckReqd := 1, Cfg_TransitStallAckReqd := 1, Cfg_IntlkTripAckReqd := 1, Cfg_IOFaultAckReqd := 1, Cfg_FullStallSeverity := 1000, Cfg_TransitStallSeverity := 1000, Cfg_IntlkTripSeverity := 500, Cfg_IOFaultSeverity := 1000, Cfg_FullStallT := 5, Cfg_TransitStallT := 10, PCmd_Close := 1, PCmd_Acq := 1, Out := 1, SrcQ_IO := 2, SrcQ := 2, Val_Fdbk := 1, Val_Sts := 1, Val_Mode := 8, Sts_Closed := 1, Sts_Available := 1, Sts_Prog := 1, Ack_FullStall := 1, Ack_TransitStall := 1, Ack_IntlkTrip := 1, Ack_IOFault := 1, Rdy_Bypass := 1);   // Sample strainer discharge
   Valve_XV_18_Stats : GekkoValveStat := (Inp_Closed := 1, Out_OpenCNT := 8694.0, Out_CloseCNT := 48707.0, Inp_OpenCNTSP := 50000.0, Out_CloseReached := 1);
   Valve_XV_19 : P_ValveSO := (Inp_PermOK := 1, Inp_NBPermOK := 1, Inp_IntlkOK := 1, Inp_NBIntlkOK := 1, Cfg_LSFail := 1, Cfg_ProgDefault := 1, Cfg_ShedOnFullStall := 1, Cfg_ShedOnTransitStall := 1, Cfg_ShedOnIOFault := 1, Cfg_FullStallAckReqd := 1, Cfg_IntlkTripAckReqd := 1, Cfg_IOFaultAckReqd := 1, Cfg_FullStallSeverity := 1000, Cfg_TransitStallSeverity := 1000, Cfg_IntlkTripSeverity := 500, Cfg_IOFaultSeverity := 1000, Cfg_FullStallT := 5, Cfg_TransitStallT := 10, PCmd_Close := 1, PCmd_Acq := 1, SrcQ_IO := 2, SrcQ := 2, Val_Fdbk := 1, Val_Sts := 1, Val_Mode := 8, Sts_Closed := 1, Sts_Available := 1, Sts_Prog := 1, Ack_FullStall := 1, Ack_TransitStall := 1, Ack_IntlkTrip := 1, Ack_IOFault := 1, Rdy_Bypass := 1);   // Laser window
   Valve_XV_19_Stats : GekkoValveStat := (Inp_Closed := 1, Out_OpenCNT := 5759.0, Out_CloseCNT := 33688.0, Inp_OpenCNTSP := 25000.0, Out_CloseReached := 1);
   Valve_XV_21_30 : P_ValveSO := (Inp_PermOK := 1, Inp_NBPermOK := 1, Inp_IntlkOK := 1, Inp_NBIntlkOK := 1, Cfg_LSFail := 1, Cfg_ProgDefault := 1, Cfg_ShedOnFullStall := 1, Cfg_ShedOnTransitStall := 1, Cfg_ShedOnIOFault := 1, Cfg_FullStallAckReqd := 1, Cfg_TransitStallAckReqd := 1, Cfg_IntlkTripAckReqd := 1, Cfg_IOFaultAckReqd := 1, Cfg_FullStallSeverity := 1000, Cfg_TransitStallSeverity := 1000, Cfg_IntlkTripSeverity := 500, Cfg_IOFaultSeverity := 1000, Cfg_FullStallT := 5, Cfg_TransitStallT := 10, PCmd_Open := 1, PCmd_Acq := 1, Out := 1, SrcQ_IO := 2, SrcQ := 2, Val_Fdbk := 2, Val_Sts := 2, Val_Mode := 8, Sts_Opened := 1, Sts_Available := 1, Sts_Prog := 1, Ack_FullStall := 1, Ack_TransitStall := 1, Ack_IntlkTrip := 1, Ack_IOFault := 1, Rdy_Bypass := 1);   // Sample isolation valve
   Valve_XV_21_30_Stats : GekkoValveStat := (Inp_Opened := 1, Out_OpenCNT := 646.0, Out_CloseCNT := 4597.0, Inp_OpenCNTSP := 2600.0, Out_CloseReached := 1);
   Valve_XV_30 : P_ValveSO := (Inp_PermOK := 1, Inp_NBPermOK := 1, Inp_IntlkOK := 1, Inp_NBIntlkOK := 1, Cfg_LSFail := 1, Cfg_ProgDefault := 1, Cfg_ShedOnFullStall := 1, Cfg_ShedOnTransitStall := 1, Cfg_ShedOnIOFault := 1, Cfg_FullStallAckReqd := 1, Cfg_TransitStallAckReqd := 1, Cfg_IntlkTripAckReqd := 1, Cfg_IOFaultAckReqd := 1, Cfg_FullStallSeverity := 1000, Cfg_TransitStallSeverity := 1000, Cfg_IntlkTripSeverity := 500, Cfg_IOFaultSeverity := 1000, Cfg_FullStallT := 5, Cfg_TransitStallT := 10, PCmd_Close := 1, PCmd_Acq := 1, SrcQ_IO := 2, SrcQ := 2, Val_Fdbk := 1, Val_Sts := 1, Val_Mode := 8, Sts_Closed := 1, Sts_Available := 1, Sts_Prog := 1, Ack_FullStall := 1, Ack_TransitStall := 1, Ack_IntlkTrip := 1, Ack_IOFault := 1, Rdy_Bypass := 1);   // XRF cooling valve
   Valve_XV_30_Stats : GekkoValveStat := (Inp_Closed := 1, Out_CloseCNT := 219.0, Inp_OpenCNTSP := 2600.0, Out_CloseReached := 1);
   Valve_XV_31 : P_ValveSO := (Inp_PermOK := 1, Inp_NBPermOK := 1, Inp_IntlkOK := 1, Inp_NBIntlkOK := 1, Cfg_LSFail := 1, Cfg_ProgDefault := 1, Cfg_ShedOnFullStall := 1, Cfg_ShedOnTransitStall := 1, Cfg_ShedOnIOFault := 1, Cfg_FullStallAckReqd := 1, Cfg_TransitStallAckReqd := 1, Cfg_IntlkTripAckReqd := 1, Cfg_IOFaultAckReqd := 1, Cfg_FullStallSeverity := 1000, Cfg_TransitStallSeverity := 1000, Cfg_IntlkTripSeverity := 500, Cfg_IOFaultSeverity := 1000, Cfg_FullStallT := 5, Cfg_TransitStallT := 10, PCmd_Close := 1, PCmd_Acq := 1, SrcQ_IO := 2, SrcQ := 2, Val_Fdbk := 1, Val_Sts := 1, Val_Mode := 8, Sts_Closed := 1, Sts_Available := 1, Sts_Prog := 1, Ack_FullStall := 1, Ack_TransitStall := 1, Ack_IntlkTrip := 1, Ack_IOFault := 1, Rdy_Bypass := 1);   // Sample Valve Tank 11
   Valve_XV_32 : P_ValveSO := (Inp_PermOK := 1, Inp_NBPermOK := 1, Inp_IntlkOK := 1, Inp_NBIntlkOK := 1, Cfg_LSFail := 1, Cfg_ProgDefault := 1, Cfg_ShedOnFullStall := 1, Cfg_ShedOnTransitStall := 1, Cfg_ShedOnIOFault := 1, Cfg_FullStallAckReqd := 1, Cfg_TransitStallAckReqd := 1, Cfg_IntlkTripAckReqd := 1, Cfg_IOFaultAckReqd := 1, Cfg_FullStallSeverity := 1000, Cfg_TransitStallSeverity := 1000, Cfg_IntlkTripSeverity := 500, Cfg_IOFaultSeverity := 1000, Cfg_FullStallT := 5, Cfg_TransitStallT := 10, PCmd_Close := 1, PCmd_Acq := 1, SrcQ_IO := 2, SrcQ := 2, Val_Fdbk := 1, Val_Sts := 1, Val_Mode := 8, Sts_Closed := 1, Sts_Available := 1, Sts_Prog := 1, Ack_FullStall := 1, Ack_TransitStall := 1, Ack_IntlkTrip := 1, Ack_IOFault := 1, Rdy_Bypass := 1);   // Sample Valve Tank 12
   Valve_XV_33 : P_ValveSO := (Inp_PermOK := 1, Inp_NBPermOK := 1, Inp_IntlkOK := 1, Inp_NBIntlkOK := 1, Cfg_LSFail := 1, Cfg_ProgDefault := 1, Cfg_ShedOnFullStall := 1, Cfg_ShedOnTransitStall := 1, Cfg_ShedOnIOFault := 1, Cfg_FullStallAckReqd := 1, Cfg_TransitStallAckReqd := 1, Cfg_IntlkTripAckReqd := 1, Cfg_IOFaultAckReqd := 1, Cfg_FullStallSeverity := 1000, Cfg_TransitStallSeverity := 1000, Cfg_IntlkTripSeverity := 500, Cfg_IOFaultSeverity := 1000, Cfg_FullStallT := 5, Cfg_TransitStallT := 10, PCmd_Close := 1, PCmd_Acq := 1, SrcQ_IO := 2, SrcQ := 2, Val_Fdbk := 1, Val_Sts := 1, Val_Mode := 8, Sts_Closed := 1, Sts_Available := 1, Sts_Prog := 1, Ack_FullStall := 1, Ack_TransitStall := 1, Ack_IntlkTrip := 1, Ack_IOFault := 1, Rdy_Bypass := 1);   // Sample Valve Tank 13
   Valve_XV_34 : P_ValveSO := (Inp_PermOK := 1, Inp_NBPermOK := 1, Inp_IntlkOK := 1, Inp_NBIntlkOK := 1, Cfg_LSFail := 1, Cfg_ProgDefault := 1, Cfg_ShedOnFullStall := 1, Cfg_ShedOnTransitStall := 1, Cfg_ShedOnIOFault := 1, Cfg_FullStallAckReqd := 1, Cfg_TransitStallAckReqd := 1, Cfg_IntlkTripAckReqd := 1, Cfg_IOFaultAckReqd := 1, Cfg_FullStallSeverity := 1000, Cfg_TransitStallSeverity := 1000, Cfg_IntlkTripSeverity := 500, Cfg_IOFaultSeverity := 1000, Cfg_FullStallT := 5, Cfg_TransitStallT := 10, PCmd_Close := 1, PCmd_Acq := 1, SrcQ_IO := 2, SrcQ := 2, Val_Fdbk := 1, Val_Sts := 1, Val_Mode := 8, Sts_Closed := 1, Sts_Available := 1, Sts_Prog := 1, Ack_FullStall := 1, Ack_TransitStall := 1, Ack_IntlkTrip := 1, Ack_IOFault := 1, Rdy_Bypass := 1);   // Sample Valve Tank 14
   Valve_XV_35 : P_ValveSO := (Inp_PermOK := 1, Inp_NBPermOK := 1, Inp_IntlkOK := 1, Inp_NBIntlkOK := 1, Cfg_LSFail := 1, Cfg_ProgDefault := 1, Cfg_ShedOnFullStall := 1, Cfg_ShedOnTransitStall := 1, Cfg_ShedOnIOFault := 1, Cfg_FullStallAckReqd := 1, Cfg_TransitStallAckReqd := 1, Cfg_IntlkTripAckReqd := 1, Cfg_IOFaultAckReqd := 1, Cfg_FullStallSeverity := 1000, Cfg_TransitStallSeverity := 1000, Cfg_IntlkTripSeverity := 500, Cfg_IOFaultSeverity := 1000, Cfg_FullStallT := 5, Cfg_TransitStallT := 10, PCmd_Close := 1, PCmd_Acq := 1, SrcQ_IO := 2, SrcQ := 2, Val_Fdbk := 1, Val_Sts := 1, Val_Mode := 8, Sts_Closed := 1, Sts_Available := 1, Sts_Prog := 1, Ack_FullStall := 1, Ack_TransitStall := 1, Ack_IntlkTrip := 1, Ack_IOFault := 1, Rdy_Bypass := 1);   // Sample Valve Tank 15
   Valve_XV_36 : P_ValveSO := (Inp_PermOK := 1, Inp_NBPermOK := 1, Inp_IntlkOK := 1, Inp_NBIntlkOK := 1, Cfg_LSFail := 1, Cfg_ProgDefault := 1, Cfg_ShedOnFullStall := 1, Cfg_ShedOnTransitStall := 1, Cfg_ShedOnIOFault := 1, Cfg_FullStallAckReqd := 1, Cfg_TransitStallAckReqd := 1, Cfg_IntlkTripAckReqd := 1, Cfg_IOFaultAckReqd := 1, Cfg_FullStallSeverity := 1000, Cfg_TransitStallSeverity := 1000, Cfg_IntlkTripSeverity := 500, Cfg_IOFaultSeverity := 1000, Cfg_FullStallT := 5, Cfg_TransitStallT := 10, PCmd_Close := 1, PCmd_Acq := 1, SrcQ_IO := 2, SrcQ := 2, Val_Fdbk := 1, Val_Sts := 1, Val_Mode := 8, Sts_Closed := 1, Sts_Available := 1, Sts_Prog := 1, Ack_FullStall := 1, Ack_TransitStall := 1, Ack_IntlkTrip := 1, Ack_IOFault := 1, Rdy_Bypass := 1);   // Sample Valve Tank 16
   Valve_XV_40 : P_ValveSO := (Inp_PermOK := 1, Inp_NBPermOK := 1, Inp_IntlkOK := 1, Inp_NBIntlkOK := 1, Cfg_LSFail := 1, Cfg_ProgDefault := 1, Cfg_ShedOnFullStall := 1, Cfg_ShedOnTransitStall := 1, Cfg_ShedOnIOFault := 1, Cfg_FullStallAckReqd := 1, Cfg_TransitStallAckReqd := 1, Cfg_IntlkTripAckReqd := 1, Cfg_IOFaultAckReqd := 1, Cfg_FullStallSeverity := 1000, Cfg_TransitStallSeverity := 1000, Cfg_IntlkTripSeverity := 500, Cfg_IOFaultSeverity := 1000, Cfg_FullStallT := 5, Cfg_TransitStallT := 10, PCmd_Close := 1, PCmd_Acq := 1, SrcQ_IO := 2, SrcQ := 2, Val_Fdbk := 1, Val_Sts := 1, Val_Mode := 8, Sts_Closed := 1, Sts_Available := 1, Sts_Prog := 1, Ack_FullStall := 1, Ack_TransitStall := 1, Ack_IntlkTrip := 1, Ack_IOFault := 1, Rdy_Bypass := 1);   // XRF power on valve
   XRF_RAWDINT : DINT[100];
   XV2130ClosedOnce : BOOL;
END_VAR

PROGRAM Analogs   (* main routine Main *)
VAR
   ADD_03 : FBD_MATH;
   BNOT_01 : FBD_BOOLEAN_NOT := (Out := 1);
   BOR_03 : FBD_BOOLEAN_OR := (In1 := 1, Out := 1);
   CalStep : DINT;
   CalWater : REAL := 165.17038;
   LocalSampleTank : DINT := 6;
   LookUpTable_01 : LookUpTable := (Input := 3789.0, X6 := 3786.0, X7 := 13615.0, Y7 := 5.0, X8 := 16000.0, Y8 := 10.0, X9 := 17086.0, Y9 := 15.0, X10 := 17670.0, Y10 := 20.0, Output := 0.0015260963);
   TONR_03 : FBD_TIMER := (PRE := 10000);
END_VAR

ROUTINE AnalogInputs   (* function block diagram *)
   SHEET 1   // Purge Totaliser
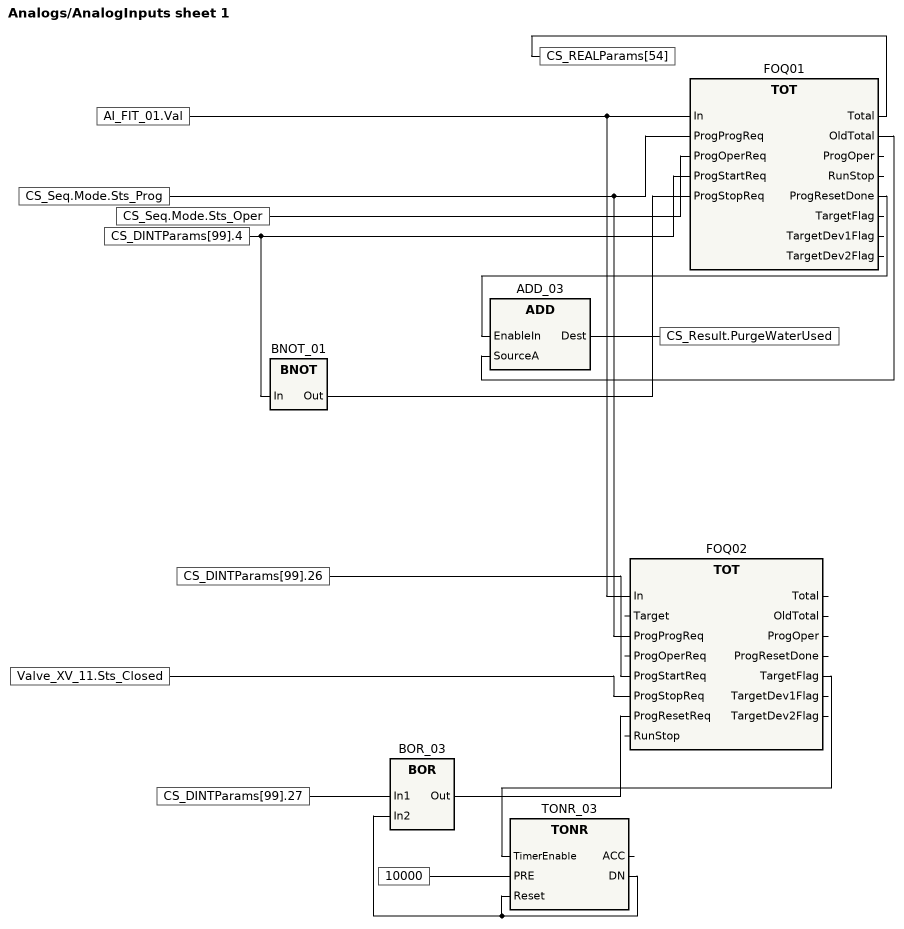
   BNOT_01 : BNOT(In := CS_DINTParams[99].4);
   BOR_03 : BOR(In1 := CS_DINTParams[99].27, In2 := TONR_03.DN {feedback});
   FOQ02 : TOT(In := AI_FIT_01.Val, ProgProgReq := CS_Seq.Mode.Sts_Prog, ProgStartReq := CS_DINTParams[99].26, ProgStopReq := Valve_XV_11.Sts_Closed, ProgResetReq := BOR_03.Out);   // unwired pins: Target ProgOperReq Total OldTotal ProgOper RunStop ProgResetDone TargetDev1Flag TargetDev2Flag
   FOQ01 : TOT(In := AI_FIT_01.Val, ProgProgReq := CS_Seq.Mode.Sts_Prog, ProgOperReq := CS_Seq.Mode.Sts_Oper, ProgStartReq := CS_DINTParams[99].4, ProgStopReq := BNOT_01.Out);   // unwired pins: ProgOper RunStop TargetFlag TargetDev1Flag TargetDev2Flag
   ADD_03 : ADD(EnableIn := FOQ01.ProgResetDone, SourceA := FOQ01.OldTotal);
   CS_REALParams[54] := FOQ01.Total;
   CS_Result.PurgeWaterUsed := ADD_03.Dest;
   TONR_03 : TONR(TimerEnable := FOQ02.TargetFlag, PRE := 10000, Reset := TONR_03.DN);   // unwired pins: ACC
END_ROUTINE

ROUTINE Analogs   (* ladder *)
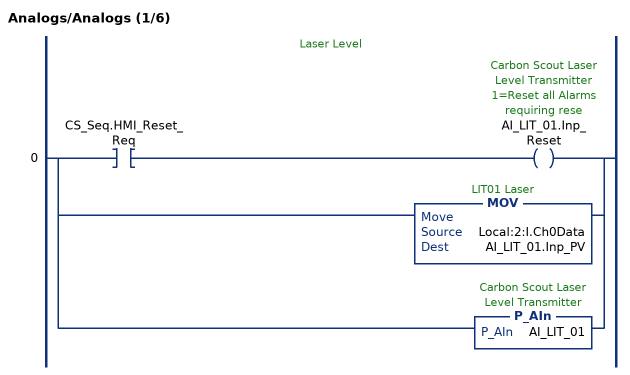
   // Laser Level
   0: [XIC(CS_Seq.HMI_Reset_Req) OTE(AI_LIT_01.Inp_Reset) ,MOV(Local:2:I.Ch0Data,AI_LIT_01.Inp_PV) ,P_AIn(AI_LIT_01) ];
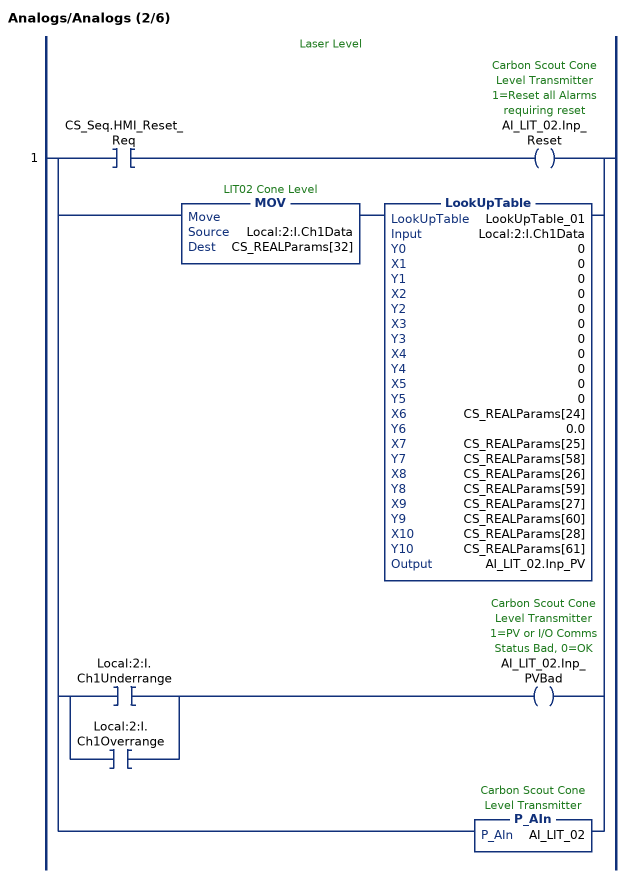
   // Laser Level
   1: [XIC(CS_Seq.HMI_Reset_Req) OTE(AI_LIT_02.Inp_Reset) ,MOV(Local:2:I.Ch1Data,CS_REALParams[32]) LookUpTable(LookUpTable_01,Local:2:I.Ch1Data,0,0,0,0,0,0,0,0,0,0,0,CS_REALParams[24],0.0,CS_REALParams[25],CS_REALParams[58],CS_REALParams[26],CS_REALParams[59],CS_REALParams[27],CS_REALParams[60],CS_REALParams[28],CS_REALParams[61],AI_LIT_02.Inp_PV) ,[XIC(Local:2:I.Ch1Underrange) ,XIC(Local:2:I.Ch1Overrange) ] OTE(AI_LIT_02.Inp_PVBad) ,P_AIn(AI_LIT_02) ];
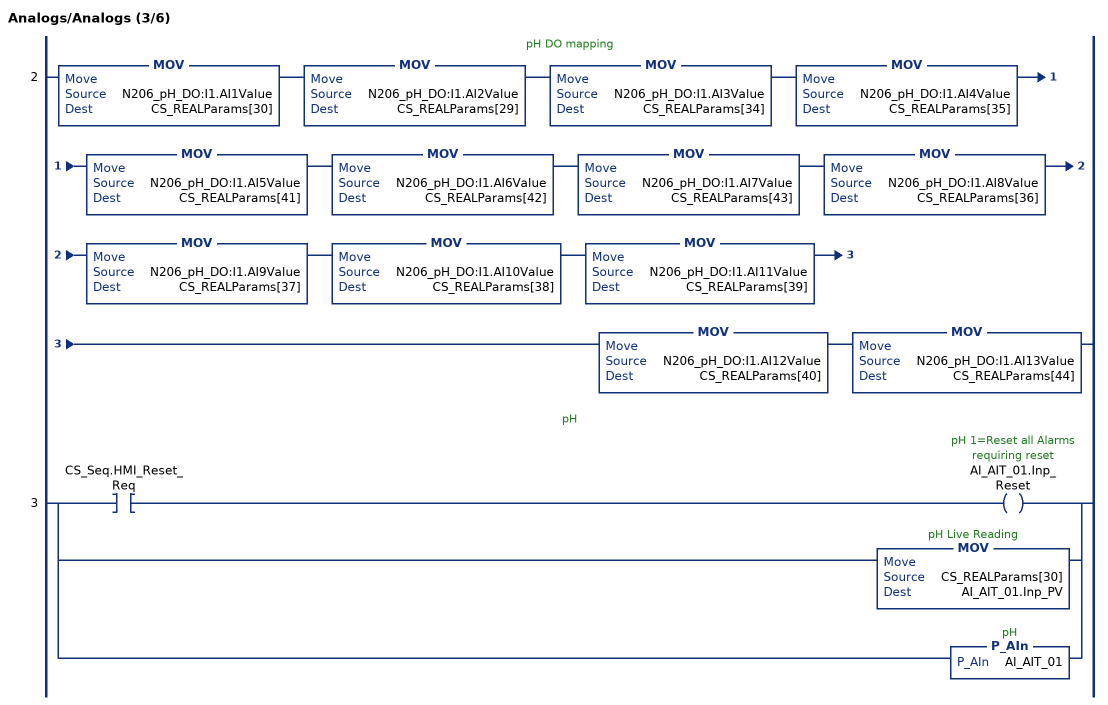
   // pH DO mapping
   2: MOV(N206_pH_DO:I1.AI1Value,CS_REALParams[30])MOV(N206_pH_DO:I1.AI2Value,CS_REALParams[29])MOV(N206_pH_DO:I1.AI3Value,CS_REALParams[34])MOV(N206_pH_DO:I1.AI4Value,CS_REALParams[35])MOV(N206_pH_DO:I1.AI5Value,CS_REALParams[41])MOV(N206_pH_DO:I1.AI6Value,CS_REALParams[42])MOV(N206_pH_DO:I1.AI7Value,CS_REALParams[43])MOV(N206_pH_DO:I1.AI8Value,CS_REALParams[36])MOV(N206_pH_DO:I1.AI9Value,CS_REALParams[37])MOV(N206_pH_DO:I1.AI10Value,CS_REALParams[38])MOV(N206_pH_DO:I1.AI11Value,CS_REALParams[39])MOV(N206_pH_DO:I1.AI12Value,CS_REALParams[40])MOV(N206_pH_DO:I1.AI13Value,CS_REALParams[44]);
   // pH
   3: [XIC(CS_Seq.HMI_Reset_Req) OTE(AI_AIT_01.Inp_Reset) ,MOV(CS_REALParams[30],AI_AIT_01.Inp_PV) ,P_AIn(AI_AIT_01) ];
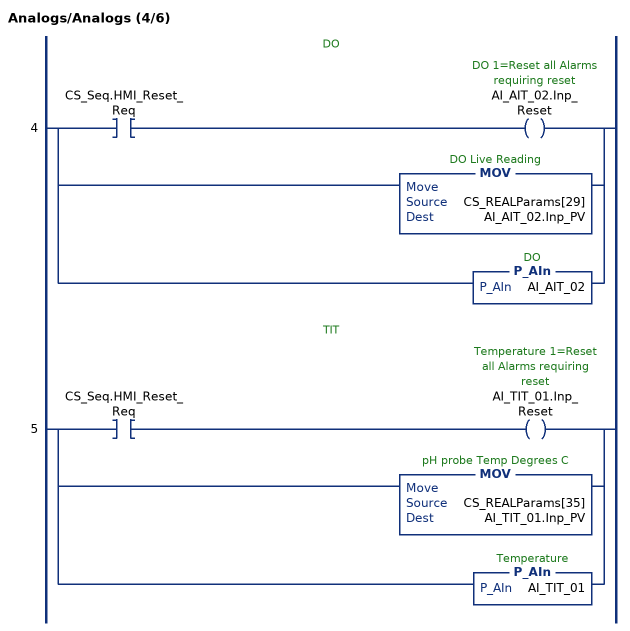
   // DO
   4: [XIC(CS_Seq.HMI_Reset_Req) OTE(AI_AIT_02.Inp_Reset) ,MOV(CS_REALParams[29],AI_AIT_02.Inp_PV) ,P_AIn(AI_AIT_02) ];
   // TIT
   5: [XIC(CS_Seq.HMI_Reset_Req) OTE(AI_TIT_01.Inp_Reset) ,MOV(CS_REALParams[35],AI_TIT_01.Inp_PV) ,P_AIn(AI_TIT_01) ];
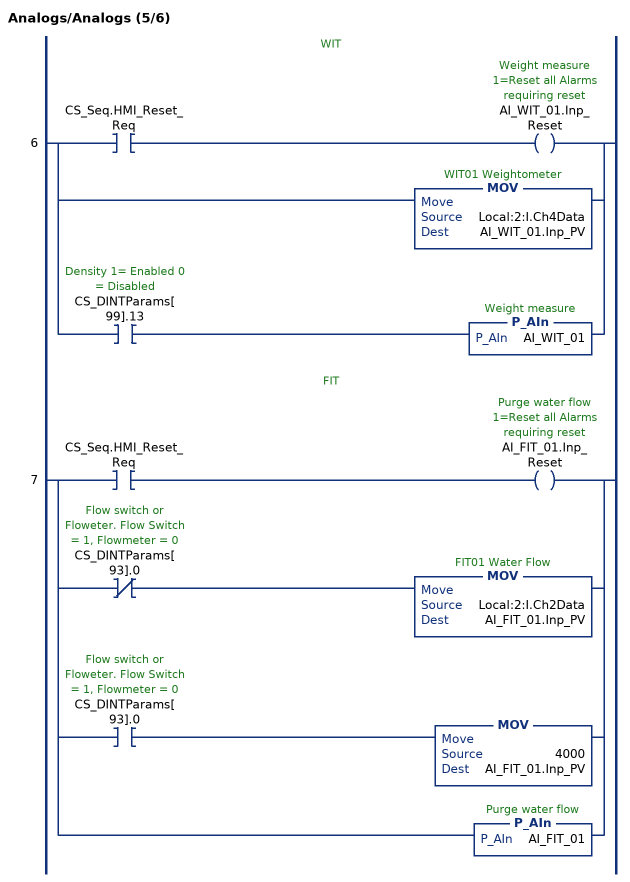
   // WIT
   6: [XIC(CS_Seq.HMI_Reset_Req) OTE(AI_WIT_01.Inp_Reset) ,MOV(Local:2:I.Ch4Data,AI_WIT_01.Inp_PV) ,XIC(CS_DINTParams[99].13) P_AIn(AI_WIT_01) ];
   // FIT
   7: [XIC(CS_Seq.HMI_Reset_Req) OTE(AI_FIT_01.Inp_Reset) ,[XIO(CS_DINTParams[93].0) MOV(Local:2:I.Ch2Data,AI_FIT_01.Inp_PV) ,XIC(CS_DINTParams[93].0) MOV(4000,AI_FIT_01.Inp_PV) ] ,P_AIn(AI_FIT_01) ];
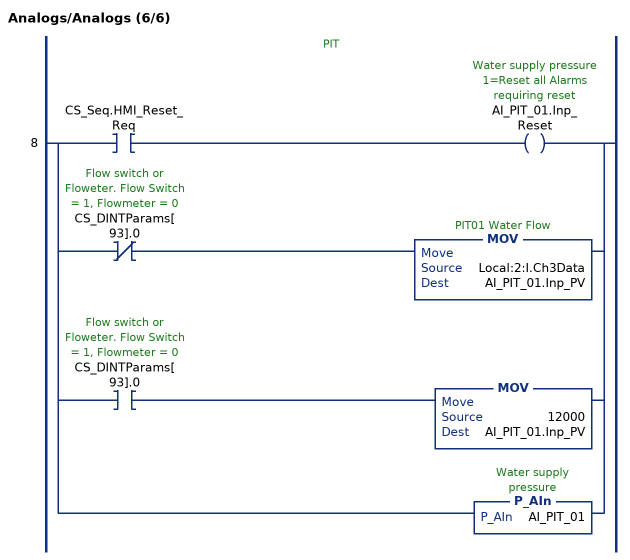
   // PIT
   8: [XIC(CS_Seq.HMI_Reset_Req) OTE(AI_PIT_01.Inp_Reset) ,[XIO(CS_DINTParams[93].0) MOV(Local:2:I.Ch3Data,AI_PIT_01.Inp_PV) ,XIC(CS_DINTParams[93].0) MOV(12000,AI_PIT_01.Inp_PV) ] ,P_AIn(AI_PIT_01) ];
END_ROUTINE

ROUTINE Main   (* ladder *)
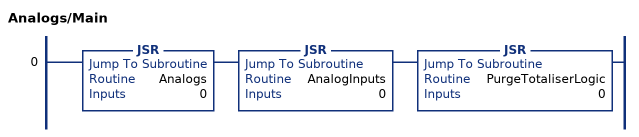
   0: JSR(Analogs,0)JSR(AnalogInputs,0)JSR(PurgeTotaliserLogic,0);
END_ROUTINE

ROUTINE PurgeTotaliserLogic   (* ladder *)
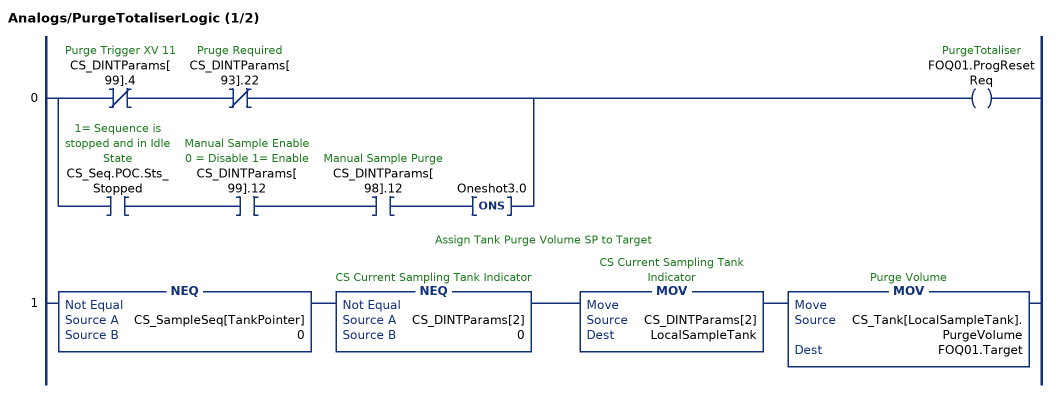
   0: [XIO(CS_DINTParams[99].4) XIO(CS_DINTParams[93].22) ,XIC(CS_Seq.POC.Sts_Stopped) XIC(CS_DINTParams[99].12) XIC(CS_DINTParams[98].12) ONS(Oneshot3.0) ]OTE(FOQ01.ProgResetReq);
   // Assign Tank Purge Volume SP to Target
   1: NEQ(CS_SampleSeq[TankPointer],0)NEQ(CS_DINTParams[2],0)MOV(CS_DINTParams[2],LocalSampleTank)MOV(CS_Tank[LocalSampleTank].PurgeVolume,FOQ01.Target);
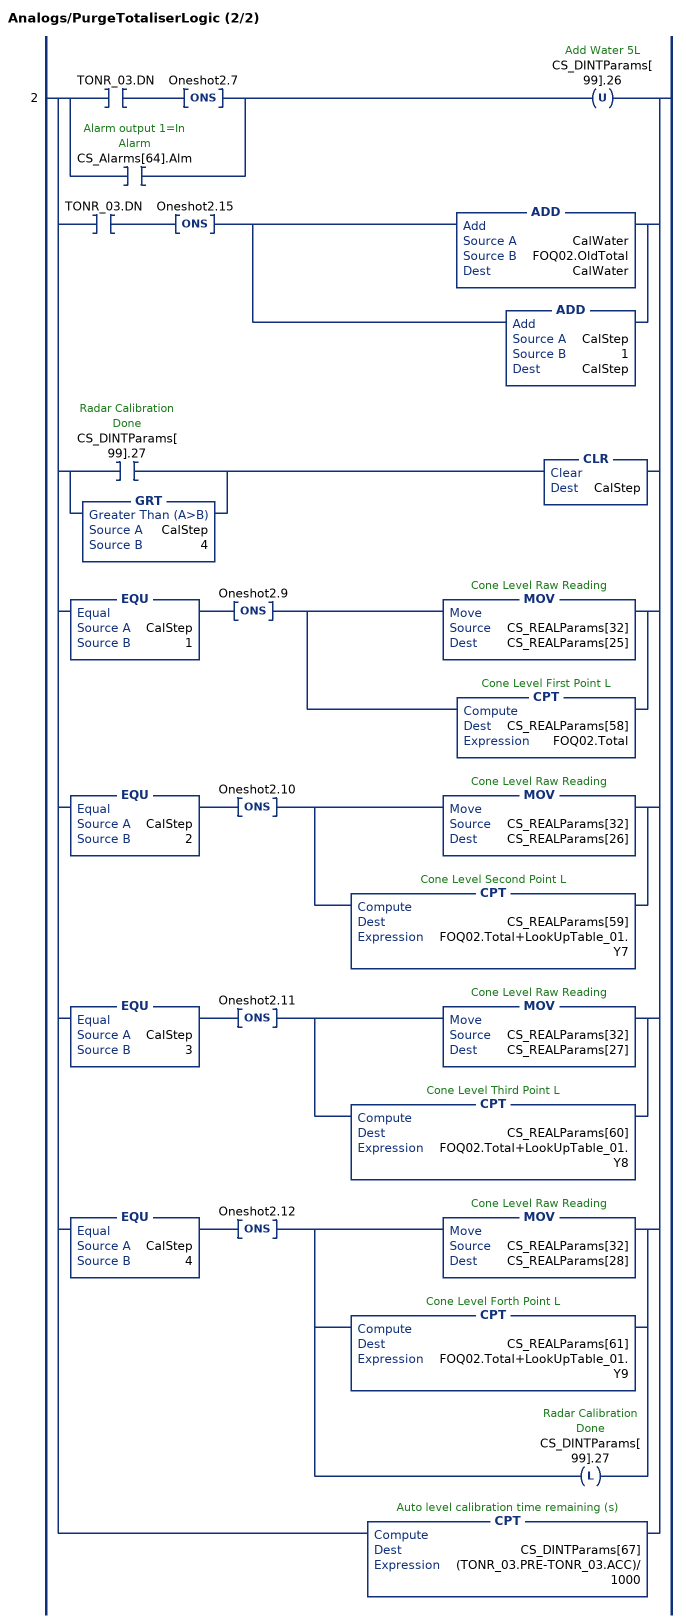
   2: [[XIC(TONR_03.DN) ONS(Oneshot2.7) ,XIC(CS_Alarms[64].Alm) ] OTU(CS_DINTParams[99].26) ,XIC(TONR_03.DN) ONS(Oneshot2.15) [ADD(CalWater,FOQ02.OldTotal,CalWater) ,ADD(CalStep,1,CalStep) ] ,[XIC(CS_DINTParams[99].27) ,GRT(CalStep,4) ] CLR(CalStep) ,EQU(CalStep,1) ONS(Oneshot2.9) [MOV(CS_REALParams[32],CS_REALParams[25]) ,CPT(CS_REALParams[58],FOQ02.Total) ] ,EQU(CalStep,2) ONS(Oneshot2.10) [MOV(CS_REALParams[32],CS_REALParams[26]) ,CPT(CS_REALParams[59],FOQ02.Total+LookUpTable_01.Y7) ] ,EQU(CalStep,3) ONS(Oneshot2.11) [MOV(CS_REALParams[32],CS_REALParams[27]) ,CPT(CS_REALParams[60],FOQ02.Total+LookUpTable_01.Y8) ] ,EQU(CalStep,4) ONS(Oneshot2.12) [MOV(CS_REALParams[32],CS_REALParams[28]) ,CPT(CS_REALParams[61],FOQ02.Total+LookUpTable_01.Y9) ,OTL(CS_DINTParams[99].27) ] ,CPT(CS_DINTParams[67],(TONR_03.PRE-TONR_03.ACC)/1000) ];
END_ROUTINE
END_PROGRAM

PROGRAM DataMapping   (* main routine Main *)
VAR
   LONS : DINT; {access Read Only}
   Oneshot4 : DINT;
END_VAR

ROUTINE DataMap   (* ladder *)
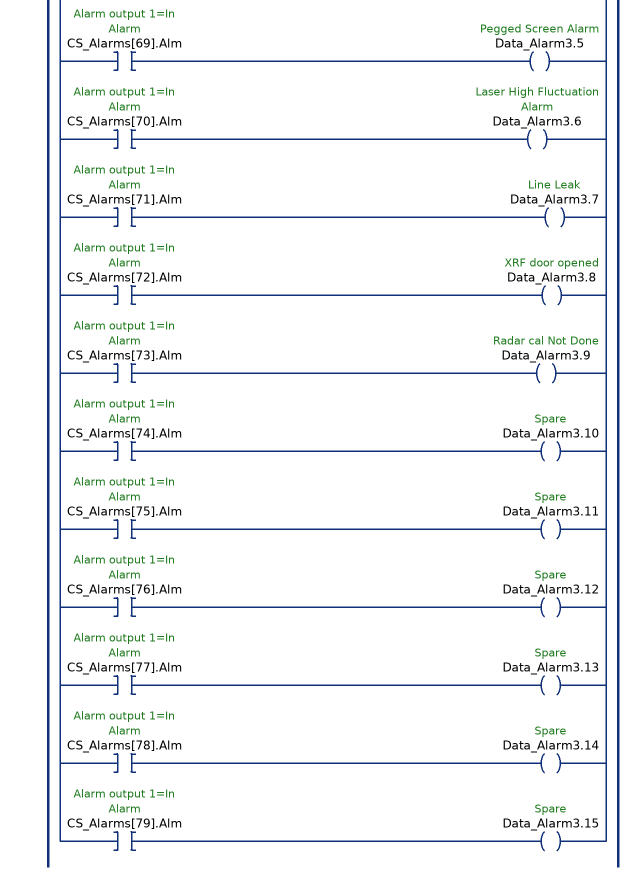
   // Alarms
   0: [XIC(CS_Alarms[0].Alm) OTE(Data_Alarm1.0) ,XIC(CS_Alarms[1].Alm) OTE(Data_Alarm1.1) ,XIC(CS_Alarms[2].Alm) OTE(Data_Alarm1.2) ,XIC(CS_Alarms[3].Alm) OTE(Data_Alarm1.3) ,XIC(CS_Alarms[4].Alm) OTE(Data_Alarm1.4) ,XIC(CS_Alarms[5].Alm) OTE(Data_Alarm1.5) ,XIC(CS_Alarms[6].Alm) OTE(Data_Alarm1.6) ,XIC(CS_Alarms[7].Alm) OTE(Data_Alarm1.7) ,XIC(CS_Alarms[8].Alm) OTE(Data_Alarm1.8) ,XIC(CS_Alarms[9].Alm) OTE(Data_Alarm1.9) ,XIC(CS_Alarms[10].Alm) OTE(Data_Alarm1.10) ,XIC(CS_Alarms[11].Alm) OTE(Data_Alarm1.11) ,XIC(CS_Alarms[12].Alm) OTE(Data_Alarm1.12) ,XIC(CS_Alarms[13].Alm) OTE(Data_Alarm1.13) ,XIC(CS_Alarms[14].Alm) OTE(Data_Alarm1.14) ,XIC(CS_Alarms[15].Alm) OTE(Data_Alarm1.15) ,XIC(CS_Alarms[16].Alm) OTE(Data_Alarm1.16) ,XIC(CS_Alarms[17].Alm) OTE(Data_Alarm1.17) ,XIC(CS_Alarms[18].Alm) OTE(Data_Alarm1.18) ,XIC(CS_Alarms[19].Alm) OTE(Data_Alarm1.19) ,XIC(CS_Alarms[20].Alm) OTE(Data_Alarm1.20) ,XIC(CS_Alarms[21].Alm) OTE(Data_Alarm1.21) ,XIC(CS_Alarms[22].Alm) OTE(Data_Alarm1.22) ,XIC(CS_Alarms[23].Alm) OTE(Data_Alarm1.23) ,XIC(CS_Alarms[24].Alm) OTE(Data_Alarm1.24) ,XIC(CS_Alarms[25].Alm) OTE(Data_Alarm1.25) ,XIC(CS_Alarms[26].Alm) OTE(Data_Alarm1.26) ,XIC(CS_Alarms[27].Alm) OTE(Data_Alarm1.27) ,XIC(CS_Alarms[31].Alm) OTE(Data_Alarm1.28) ,XIC(CS_Alarms[29].Alm) OTE(Data_Alarm1.29) ,XIC(CS_Alarms[30].Alm) OTE(Data_Alarm1.30) ,AFI() OTE(Data_Alarm1.31) ,XIC(CS_Alarms[32].Alm) OTE(Data_Alarm2.0) ,XIC(CS_Alarms[33].Alm) OTE(Data_Alarm2.1) ,XIC(CS_Alarms[34].Alm) OTE(Data_Alarm2.2) ,XIC(CS_Alarms[35].Alm) OTE(Data_Alarm2.3) ,XIC(CS_Alarms[36].Alm) OTE(Data_Alarm2.4) ,XIC(CS_Alarms[37].Alm) OTE(Data_Alarm2.5) ,XIC(CS_Alarms[38].Alm) OTE(Data_Alarm2.6) ,XIC(CS_Alarms[39].Alm) OTE(Data_Alarm2.7) ,XIC(CS_Alarms[40].Alm) OTE(Data_Alarm2.8) ,XIC(CS_Alarms[41].Alm) OTE(Data_Alarm2.9) ,XIC(CS_Alarms[42].Alm) OTE(Data_Alarm2.10) ,XIC(CS_Alarms[43].Alm) OTE(Data_Alarm2.11) ,XIC(CS_Alarms[63].Alm) OTE(Data_Alarm2.12) ,XIC(CS_Alarms[45].Alm) OTE(Data_Alarm2.13) ,XIC(CS_Alarms[46].Alm) OTE(Data_Alarm2.14) ,XIC(CS_Alarms[47].Alm) OTE(Data_Alarm2.15) ,XIC(CS_Alarms[48].Alm) OTE(Data_Alarm2.16) ,XIC(CS_Alarms[49].Alm) OTE(Data_Alarm2.17) ,XIC(CS_Alarms[50].Alm) OTE(Data_Alarm2.18) ,XIC(CS_Alarms[51].Alm) OTE(Data_Alarm2.19) ,XIC(CS_Alarms[52].Alm) OTE(Data_Alarm2.20) ,XIC(CS_Alarms[53].Alm) OTE(Data_Alarm2.21) ,XIC(CS_Alarms[54].Alm) OTE(Data_Alarm2.22) ,XIC(CS_Alarms[55].Alm) OTE(Data_Alarm2.23) ,XIC(CS_Alarms[56].Alm) OTE(Data_Alarm2.24) ,XIC(CS_Alarms[57].Alm) OTE(Data_Alarm2.25) ,XIC(CS_Alarms[58].Alm) OTE(Data_Alarm2.26) ,XIC(CS_Alarms[59].Alm) OTE(Data_Alarm2.27) ,XIC(CS_Alarms[60].Alm) OTE(Data_Alarm2.28) ,XIC(CS_Alarms[61].Alm) OTE(Data_Alarm2.29) ,XIC(CS_Alarms[62].Alm) OTE(Data_Alarm2.30) ,AFI() OTE(Data_Alarm2.31) ,XIC(CS_Alarms[64].Alm) OTE(Data_Alarm3.0) ,XIC(CS_Alarms[65].Alm) OTE(Data_Alarm3.1) ,XIC(CS_Alarms[66].Alm) OTE(Data_Alarm3.2) ,XIC(CS_Alarms[67].Alm) OTE(Data_Alarm3.3) ,XIC(CS_Alarms[68].Alm) OTE(Data_Alarm3.4) ,XIC(CS_Alarms[69].Alm) OTE(Data_Alarm3.5) ,XIC(CS_Alarms[70].Alm) OTE(Data_Alarm3.6) ,XIC(CS_Alarms[71].Alm) OTE(Data_Alarm3.7) ,XIC(CS_Alarms[72].Alm) OTE(Data_Alarm3.8) ,XIC(CS_Alarms[73].Alm) OTE(Data_Alarm3.9) ,XIC(CS_Alarms[74].Alm) OTE(Data_Alarm3.10) ,XIC(CS_Alarms[75].Alm) OTE(Data_Alarm3.11) ,XIC(CS_Alarms[76].Alm) OTE(Data_Alarm3.12) ,XIC(CS_Alarms[77].Alm) OTE(Data_Alarm3.13) ,XIC(CS_Alarms[78].Alm) OTE(Data_Alarm3.14) ,XIC(CS_Alarms[79].Alm) OTE(Data_Alarm3.15) ];
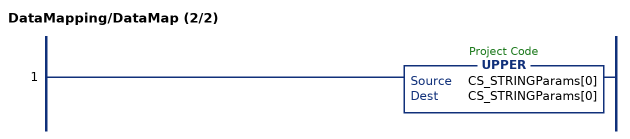
   1: UPPER(CS_STRINGParams[0],CS_STRINGParams[0]);
END_ROUTINE

ROUTINE DCSMapping   (* ladder *)
// Maintain data connection with old program tags
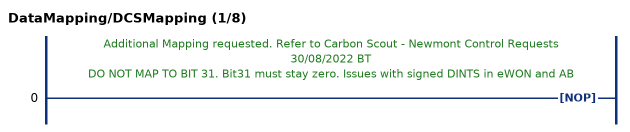
   // Additional Mapping requested. Refer to Carbon Scout - Newmont Control Requests 30/08/2022 BT
   // DO NOT MAP TO BIT 31. Bit31 must stay zero. Issues with signed DINTS in eWON and AB
   0: NOP();
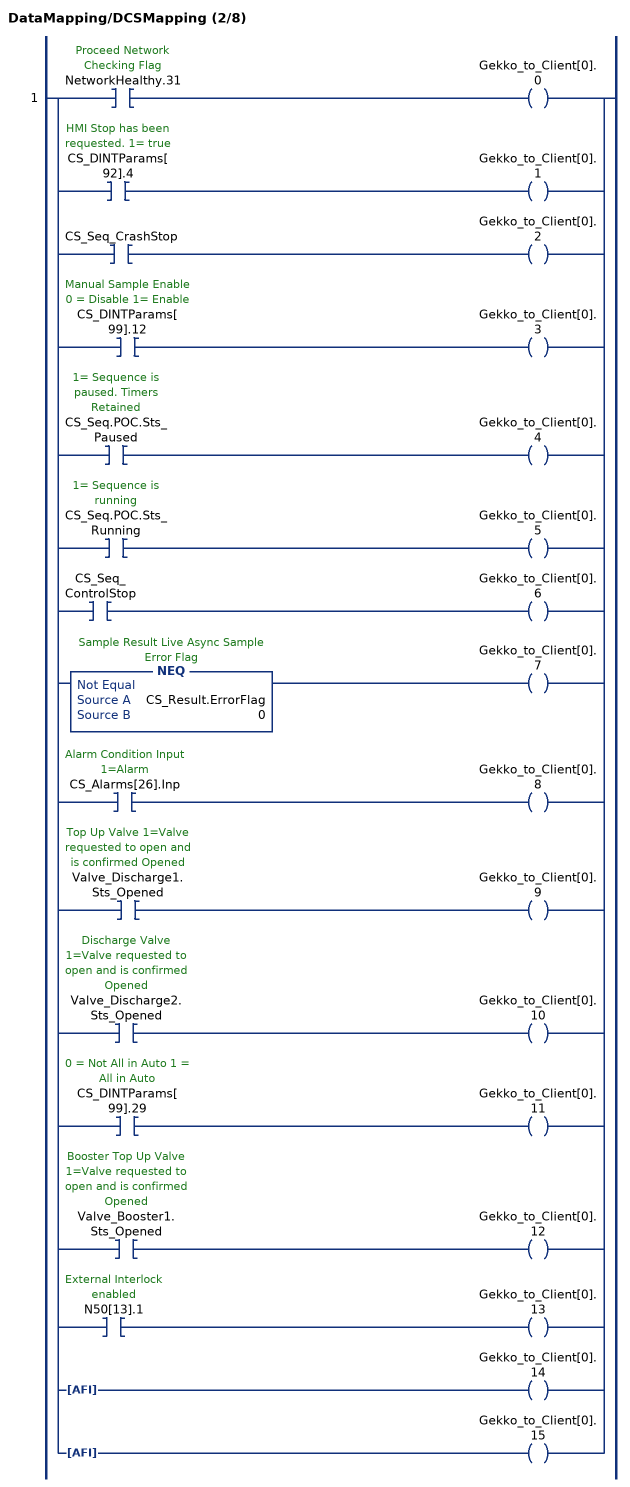
   1: [XIC(NetworkHealthy.31) OTE(Gekko_to_Client[0].0) ,XIC(CS_DINTParams[92].4) OTE(Gekko_to_Client[0].1) ,XIC(CS_Seq_CrashStop) OTE(Gekko_to_Client[0].2) ,XIC(CS_DINTParams[99].12) OTE(Gekko_to_Client[0].3) ,XIC(CS_Seq.POC.Sts_Paused) OTE(Gekko_to_Client[0].4) ,XIC(CS_Seq.POC.Sts_Running) OTE(Gekko_to_Client[0].5) ,XIC(CS_Seq_ControlStop) OTE(Gekko_to_Client[0].6) ,NEQ(CS_Result.ErrorFlag,0) OTE(Gekko_to_Client[0].7) ,XIC(CS_Alarms[26].Inp) OTE(Gekko_to_Client[0].8) ,XIC(Valve_Discharge1.Sts_Opened) OTE(Gekko_to_Client[0].9) ,XIC(Valve_Discharge2.Sts_Opened) OTE(Gekko_to_Client[0].10) ,XIC(CS_DINTParams[99].29) OTE(Gekko_to_Client[0].11) ,XIC(Valve_Booster1.Sts_Opened) OTE(Gekko_to_Client[0].12) ,XIC(N50[13].1) OTE(Gekko_to_Client[0].13) ,AFI() OTE(Gekko_to_Client[0].14) ,AFI() OTE(Gekko_to_Client[0].15) ];
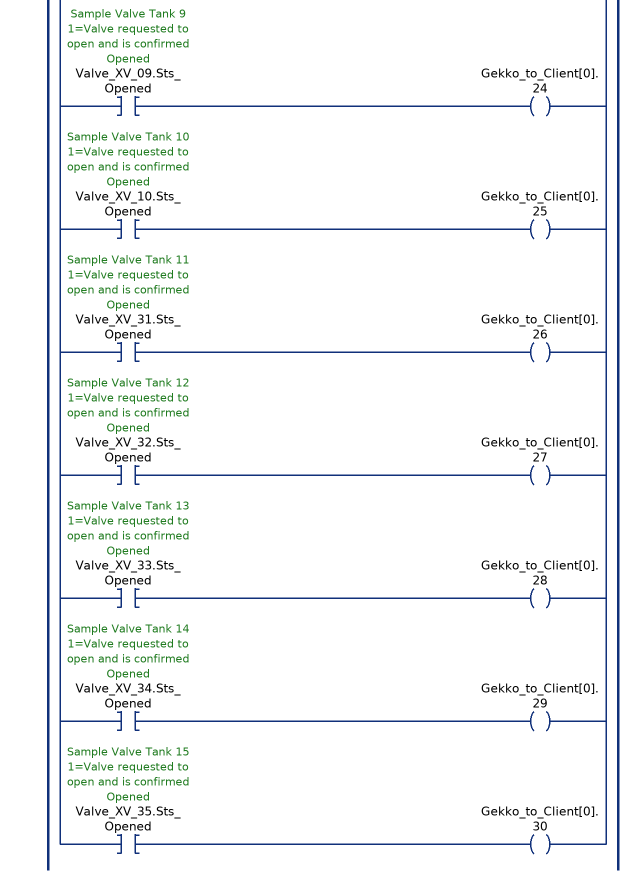
   2: [XIC(Valve_XV_01.Sts_Opened) OTE(Gekko_to_Client[0].16) ,XIC(Valve_XV_02.Sts_Opened) OTE(Gekko_to_Client[0].17) ,XIC(Valve_XV_03.Sts_Opened) OTE(Gekko_to_Client[0].18) ,XIC(Valve_XV_04.Sts_Opened) OTE(Gekko_to_Client[0].19) ,XIC(Valve_XV_05.Sts_Opened) OTE(Gekko_to_Client[0].20) ,XIC(Valve_XV_06.Sts_Opened) OTE(Gekko_to_Client[0].21) ,XIC(Valve_XV_07.Sts_Opened) OTE(Gekko_to_Client[0].22) ,XIC(Valve_XV_08.Sts_Opened) OTE(Gekko_to_Client[0].23) ,XIC(Valve_XV_09.Sts_Opened) OTE(Gekko_to_Client[0].24) ,XIC(Valve_XV_10.Sts_Opened) OTE(Gekko_to_Client[0].25) ,XIC(Valve_XV_31.Sts_Opened) OTE(Gekko_to_Client[0].26) ,XIC(Valve_XV_32.Sts_Opened) OTE(Gekko_to_Client[0].27) ,XIC(Valve_XV_33.Sts_Opened) OTE(Gekko_to_Client[0].28) ,XIC(Valve_XV_34.Sts_Opened) OTE(Gekko_to_Client[0].29) ,XIC(Valve_XV_35.Sts_Opened) OTE(Gekko_to_Client[0].30) ];
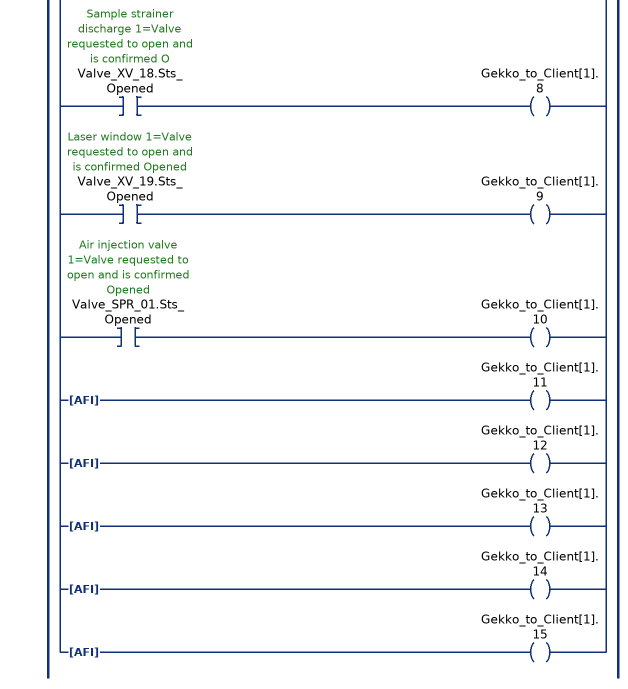
   3: [XIC(Valve_XV_36.Sts_Opened) OTE(Gekko_to_Client[1].0) ,XIC(Valve_XV_11.Sts_Opened) OTE(Gekko_to_Client[1].1) ,XIC(Valve_XV_12.Sts_Opened) OTE(Gekko_to_Client[1].2) ,XIC(Valve_XV_13.Sts_Opened) OTE(Gekko_to_Client[1].3) ,XIC(Valve_XV_14.Sts_Opened) OTE(Gekko_to_Client[1].4) ,XIC(Valve_XV_15.Sts_Opened) OTE(Gekko_to_Client[1].5) ,XIC(Valve_XV_16.Sts_Opened) OTE(Gekko_to_Client[1].6) ,XIC(Valve_XV_17.Sts_Opened) OTE(Gekko_to_Client[1].7) ,XIC(Valve_XV_18.Sts_Opened) OTE(Gekko_to_Client[1].8) ,XIC(Valve_XV_19.Sts_Opened) OTE(Gekko_to_Client[1].9) ,XIC(Valve_SPR_01.Sts_Opened) OTE(Gekko_to_Client[1].10) ,AFI() OTE(Gekko_to_Client[1].11) ,AFI() OTE(Gekko_to_Client[1].12) ,AFI() OTE(Gekko_to_Client[1].13) ,AFI() OTE(Gekko_to_Client[1].14) ,AFI() OTE(Gekko_to_Client[1].15) ];
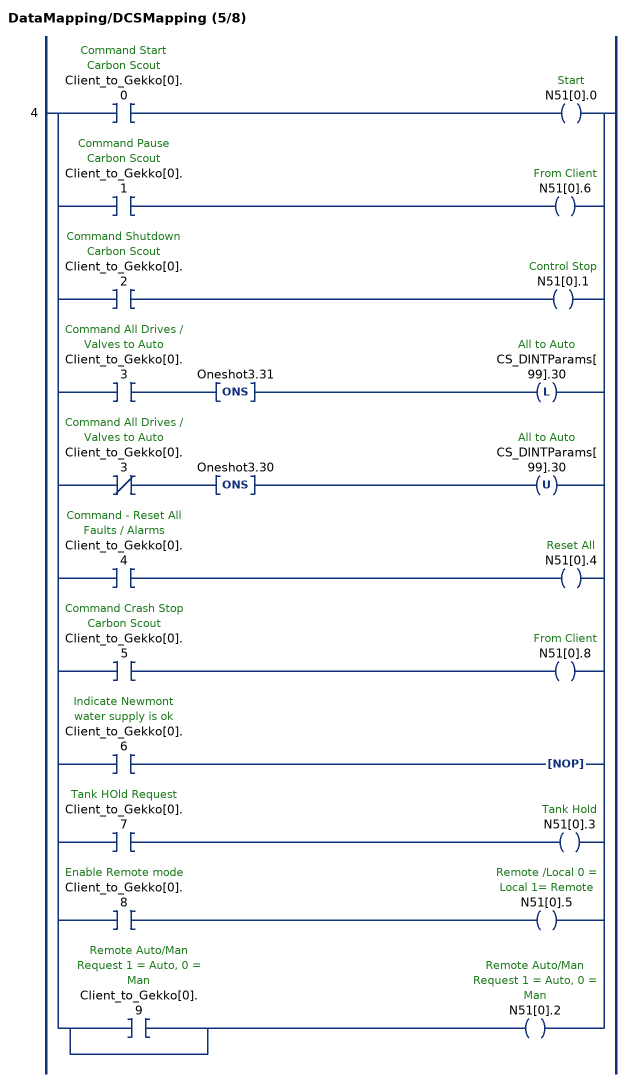
   4: [XIC(Client_to_Gekko[0].0) OTE(N51[0].0) ,XIC(Client_to_Gekko[0].1) OTE(N51[0].6) ,XIC(Client_to_Gekko[0].2) OTE(N51[0].1) ,[XIC(Client_to_Gekko[0].3) ONS(Oneshot3.31) OTL(CS_DINTParams[99].30) ,XIO(Client_to_Gekko[0].3) ONS(Oneshot3.30) OTU(CS_DINTParams[99].30) ] ,XIC(Client_to_Gekko[0].4) OTE(N51[0].4) ,XIC(Client_to_Gekko[0].5) OTE(N51[0].8) ,XIC(Client_to_Gekko[0].6) NOP() ,XIC(Client_to_Gekko[0].7) OTE(N51[0].3) ,XIC(Client_to_Gekko[0].8) OTE(N51[0].5) ,[XIC(Client_to_Gekko[0].9) ,] OTE(N51[0].2) ];
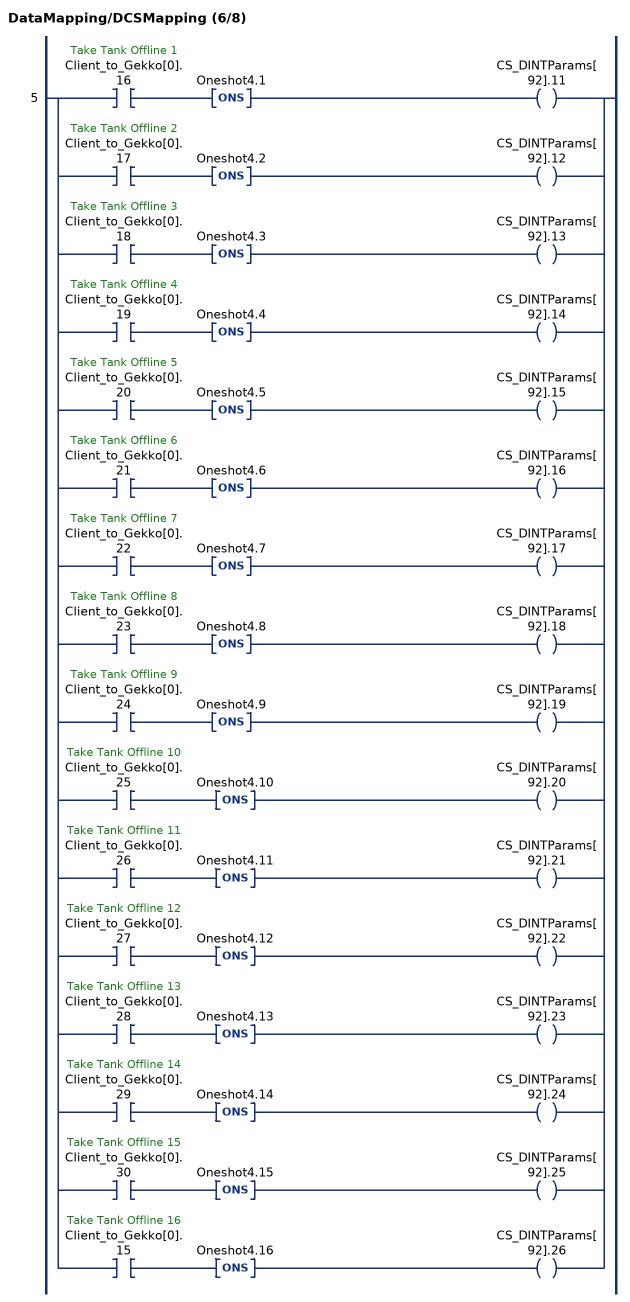
   5: [XIC(Client_to_Gekko[0].16) ONS(Oneshot4.1) OTE(CS_DINTParams[92].11) ,XIC(Client_to_Gekko[0].17) ONS(Oneshot4.2) OTE(CS_DINTParams[92].12) ,XIC(Client_to_Gekko[0].18) ONS(Oneshot4.3) OTE(CS_DINTParams[92].13) ,XIC(Client_to_Gekko[0].19) ONS(Oneshot4.4) OTE(CS_DINTParams[92].14) ,XIC(Client_to_Gekko[0].20) ONS(Oneshot4.5) OTE(CS_DINTParams[92].15) ,XIC(Client_to_Gekko[0].21) ONS(Oneshot4.6) OTE(CS_DINTParams[92].16) ,XIC(Client_to_Gekko[0].22) ONS(Oneshot4.7) OTE(CS_DINTParams[92].17) ,XIC(Client_to_Gekko[0].23) ONS(Oneshot4.8) OTE(CS_DINTParams[92].18) ,XIC(Client_to_Gekko[0].24) ONS(Oneshot4.9) OTE(CS_DINTParams[92].19) ,XIC(Client_to_Gekko[0].25) ONS(Oneshot4.10) OTE(CS_DINTParams[92].20) ,XIC(Client_to_Gekko[0].26) ONS(Oneshot4.11) OTE(CS_DINTParams[92].21) ,XIC(Client_to_Gekko[0].27) ONS(Oneshot4.12) OTE(CS_DINTParams[92].22) ,XIC(Client_to_Gekko[0].28) ONS(Oneshot4.13) OTE(CS_DINTParams[92].23) ,XIC(Client_to_Gekko[0].29) ONS(Oneshot4.14) OTE(CS_DINTParams[92].24) ,XIC(Client_to_Gekko[0].30) ONS(Oneshot4.15) OTE(CS_DINTParams[92].25) ,XIC(Client_to_Gekko[0].15) ONS(Oneshot4.16) OTE(CS_DINTParams[92].26) ];
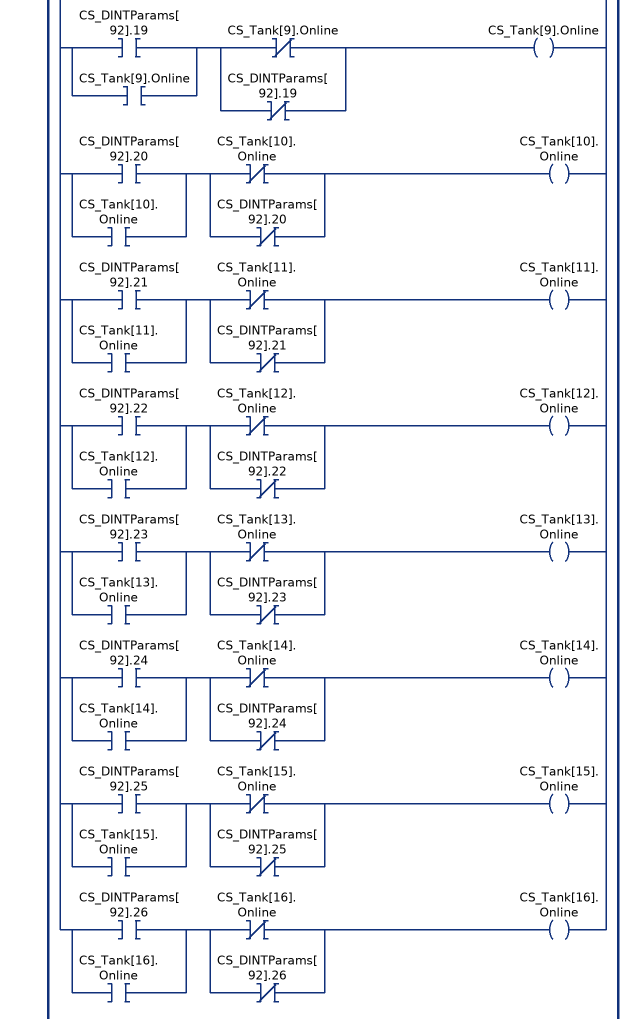
   6: [[XIC(CS_DINTParams[92].11) ,XIC(CS_Tank[1].Online) ] [XIO(CS_Tank[1].Online) ,XIO(CS_DINTParams[92].11) ] OTE(CS_Tank[1].Online) ,[XIC(CS_DINTParams[92].12) ,XIC(CS_Tank[2].Online) ] [XIO(CS_Tank[2].Online) ,XIO(CS_DINTParams[92].12) ] OTE(CS_Tank[2].Online) ,[XIC(CS_DINTParams[92].13) ,XIC(CS_Tank[3].Online) ] [XIO(CS_Tank[3].Online) ,XIO(CS_DINTParams[92].13) ] OTE(CS_Tank[3].Online) ,[XIC(CS_DINTParams[92].14) ,XIC(CS_Tank[4].Online) ] [XIO(CS_Tank[4].Online) ,XIO(CS_DINTParams[92].14) ] OTE(CS_Tank[4].Online) ,[XIC(CS_DINTParams[92].15) ,XIC(CS_Tank[5].Online) ] [XIO(CS_Tank[5].Online) ,XIO(CS_DINTParams[92].15) ] OTE(CS_Tank[5].Online) ,[XIC(CS_DINTParams[92].16) ,XIC(CS_Tank[6].Online) ] [XIO(CS_Tank[6].Online) ,XIO(CS_DINTParams[92].16) ] OTE(CS_Tank[6].Online) ,[XIC(CS_DINTParams[92].17) ,XIC(CS_Tank[7].Online) ] [XIO(CS_Tank[7].Online) ,XIO(CS_DINTParams[92].17) ] OTE(CS_Tank[7].Online) ,[XIC(CS_DINTParams[92].18) ,XIC(CS_Tank[8].Online) ] [XIO(CS_Tank[8].Online) ,XIO(CS_DINTParams[92].18) ] OTE(CS_Tank[8].Online) ,[XIC(CS_DINTParams[92].19) ,XIC(CS_Tank[9].Online) ] [XIO(CS_Tank[9].Online) ,XIO(CS_DINTParams[92].19) ] OTE(CS_Tank[9].Online) ,[XIC(CS_DINTParams[92].20) ,XIC(CS_Tank[10].Online) ] [XIO(CS_Tank[10].Online) ,XIO(CS_DINTParams[92].20) ] OTE(CS_Tank[10].Online) ,[XIC(CS_DINTParams[92].21) ,XIC(CS_Tank[11].Online) ] [XIO(CS_Tank[11].Online) ,XIO(CS_DINTParams[92].21) ] OTE(CS_Tank[11].Online) ,[XIC(CS_DINTParams[92].22) ,XIC(CS_Tank[12].Online) ] [XIO(CS_Tank[12].Online) ,XIO(CS_DINTParams[92].22) ] OTE(CS_Tank[12].Online) ,[XIC(CS_DINTParams[92].23) ,XIC(CS_Tank[13].Online) ] [XIO(CS_Tank[13].Online) ,XIO(CS_DINTParams[92].23) ] OTE(CS_Tank[13].Online) ,[XIC(CS_DINTParams[92].24) ,XIC(CS_Tank[14].Online) ] [XIO(CS_Tank[14].Online) ,XIO(CS_DINTParams[92].24) ] OTE(CS_Tank[14].Online) ,[XIC(CS_DINTParams[92].25) ,XIC(CS_Tank[15].Online) ] [XIO(CS_Tank[15].Online) ,XIO(CS_DINTParams[92].25) ] OTE(CS_Tank[15].Online) ,[XIC(CS_DINTParams[92].26) ,XIC(CS_Tank[16].Online) ] [XIO(CS_Tank[16].Online) ,XIO(CS_DINTParams[92].26) ] OTE(CS_Tank[16].Online) ];
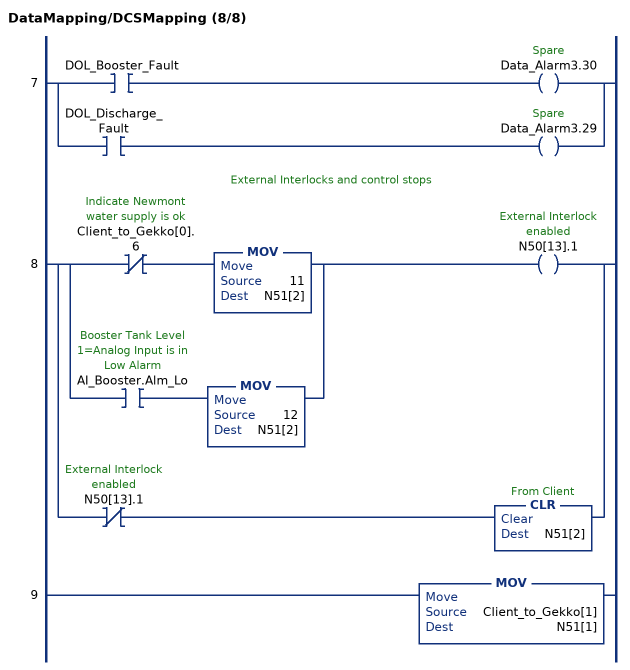
   7: [XIC(DOL_Booster_Fault) OTE(Data_Alarm3.30) ,XIC(DOL_Discharge_Fault) OTE(Data_Alarm3.29) ];
   // External Interlocks and control stops
   8: [[XIO(Client_to_Gekko[0].6) MOV(11,N51[2]) ,XIC(AI_Booster.Alm_Lo) MOV(12,N51[2]) ] OTE(N50[13].1) ,XIO(N50[13].1) CLR(N51[2]) ];
   9: MOV(Client_to_Gekko[1],N51[1]);
END_ROUTINE
